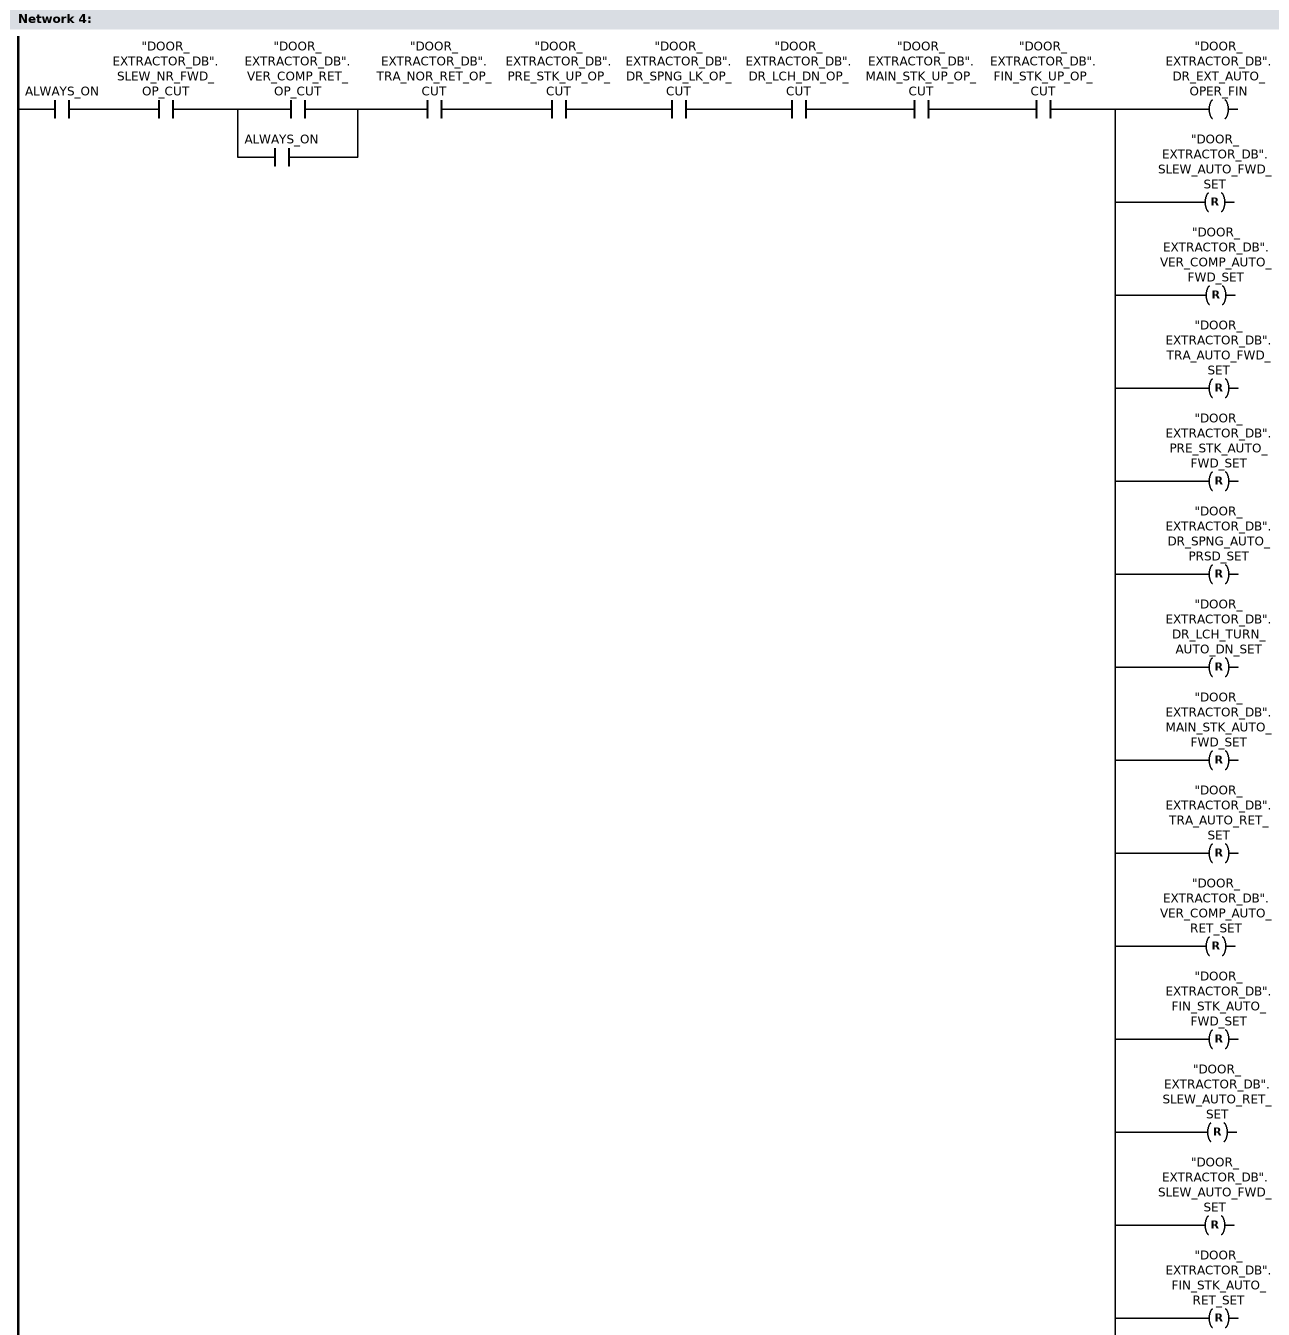
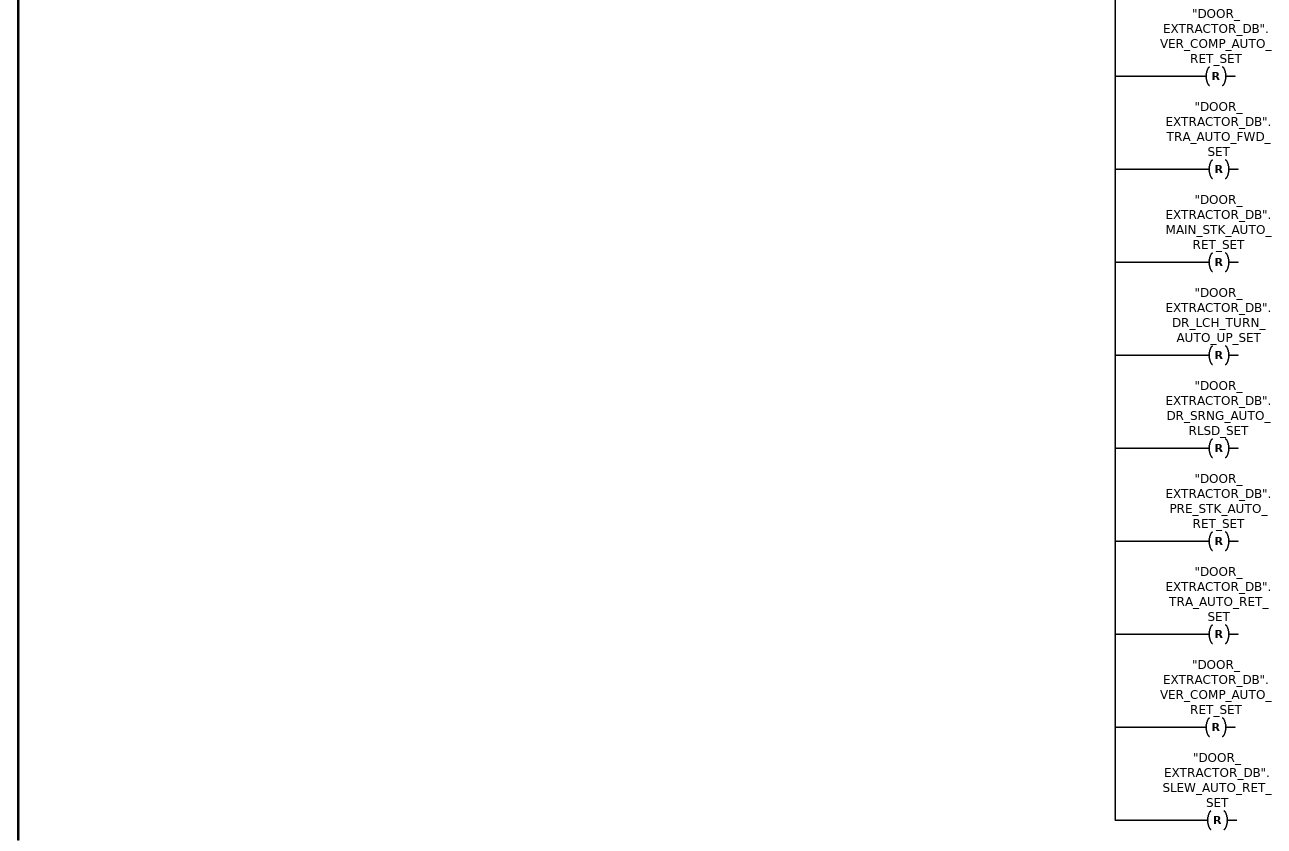
NETWORK
TITLE =
      A     "ALWAYS_ON";
      A     "DOOR_EXTRACTOR_DB".SLEW_NR_FWD_OP_CUT;
      A(;
      O     "DOOR_EXTRACTOR_DB".VER_COMP_RET_OP_CUT;
      O     "ALWAYS_ON";
      );
      A     "DOOR_EXTRACTOR_DB".TRA_NOR_RET_OP_CUT;
      A     "DOOR_EXTRACTOR_DB".PRE_STK_UP_OP_CUT;
      A     "DOOR_EXTRACTOR_DB".DR_SPNG_LK_OP_CUT;
      A     "DOOR_EXTRACTOR_DB".DR_LCH_DN_OP_CUT;
      A     "DOOR_EXTRACTOR_DB".MAIN_STK_UP_OP_CUT;
      A     "DOOR_EXTRACTOR_DB".FIN_STK_UP_OP_CUT;
      =     "DOOR_EXTRACTOR_DB".DR_EXT_AUTO_OPER_FIN;
      R     "DOOR_EXTRACTOR_DB".SLEW_AUTO_FWD_SET;
      R     "DOOR_EXTRACTOR_DB".VER_COMP_AUTO_FWD_SET;
      R     "DOOR_EXTRACTOR_DB".TRA_AUTO_FWD_SET;
      R     "DOOR_EXTRACTOR_DB".PRE_STK_AUTO_FWD_SET;
      R     "DOOR_EXTRACTOR_DB".DR_SPNG_AUTO_PRSD_SET;
      R     "DOOR_EXTRACTOR_DB".DR_LCH_TURN_AUTO_DN_SET;
      R     "DOOR_EXTRACTOR_DB".MAIN_STK_AUTO_FWD_SET;
      R     "DOOR_EXTRACTOR_DB".TRA_AUTO_RET_SET;
      R     "DOOR_EXTRACTOR_DB".VER_COMP_AUTO_RET_SET;
      R     "DOOR_EXTRACTOR_DB".FIN_STK_AUTO_FWD_SET;
      R     "DOOR_EXTRACTOR_DB".SLEW_AUTO_RET_SET;
      R     "DOOR_EXTRACTOR_DB".SLEW_AUTO_FWD_SET;
      R     "DOOR_EXTRACTOR_DB".FIN_STK_AUTO_RET_SET;
      R     "DOOR_EXTRACTOR_DB".VER_COMP_AUTO_RET_SET;
      R     "DOOR_EXTRACTOR_DB".TRA_AUTO_FWD_SET;
      R     "DOOR_EXTRACTOR_DB".MAIN_STK_AUTO_RET_SET;
      R     "DOOR_EXTRACTOR_DB".DR_LCH_TURN_AUTO_UP_SET;
      R     "DOOR_EXTRACTOR_DB".DR_SRNG_AUTO_RLSD_SET;
      R     "DOOR_EXTRACTOR_DB".PRE_STK_AUTO_RET_SET;
      R     "DOOR_EXTRACTOR_DB".TRA_AUTO_RET_SET;
      R     "DOOR_EXTRACTOR_DB".VER_COMP_AUTO_RET_SET;
      R     "DOOR_EXTRACTOR_DB".SLEW_AUTO_RET_SET;
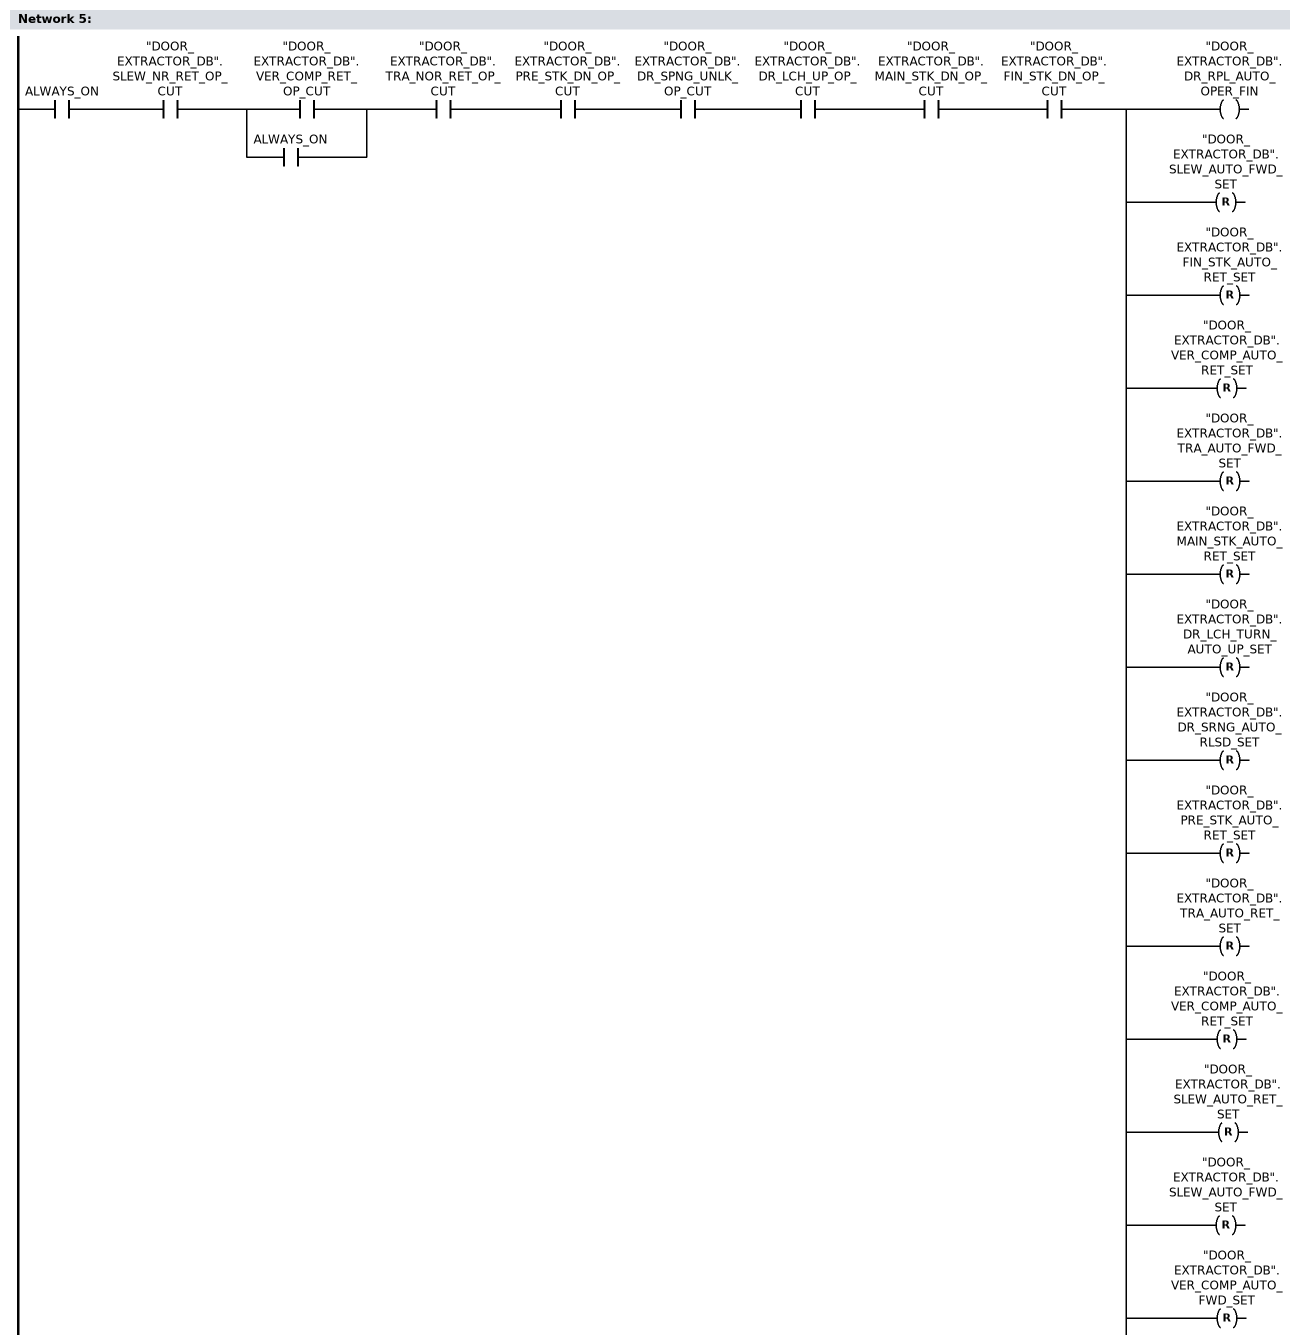
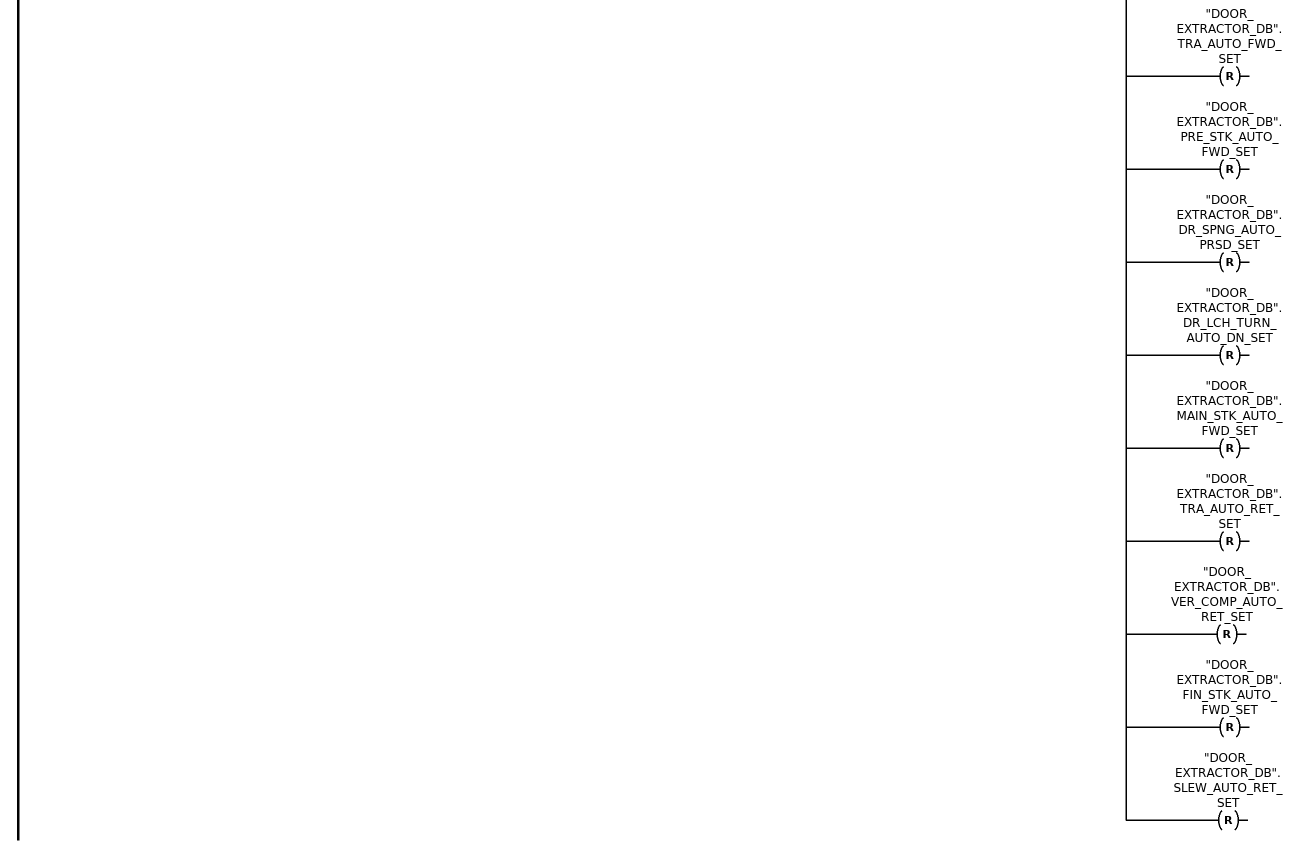
NETWORK
TITLE =
      A     "ALWAYS_ON";
      A     "DOOR_EXTRACTOR_DB".SLEW_NR_RET_OP_CUT;
      A(;
      O     "DOOR_EXTRACTOR_DB".VER_COMP_RET_OP_CUT;
      O     "ALWAYS_ON";
      );
      A     "DOOR_EXTRACTOR_DB".TRA_NOR_RET_OP_CUT;
      A     "DOOR_EXTRACTOR_DB".PRE_STK_DN_OP_CUT;
      A     "DOOR_EXTRACTOR_DB".DR_SPNG_UNLK_OP_CUT;
      A     "DOOR_EXTRACTOR_DB".DR_LCH_UP_OP_CUT;
      A     "DOOR_EXTRACTOR_DB".MAIN_STK_DN_OP_CUT;
      A     "DOOR_EXTRACTOR_DB".FIN_STK_DN_OP_CUT;
      =     "DOOR_EXTRACTOR_DB".DR_RPL_AUTO_OPER_FIN;
      R     "DOOR_EXTRACTOR_DB".SLEW_AUTO_FWD_SET;
      R     "DOOR_EXTRACTOR_DB".FIN_STK_AUTO_RET_SET;
      R     "DOOR_EXTRACTOR_DB".VER_COMP_AUTO_RET_SET;
      R     "DOOR_EXTRACTOR_DB".TRA_AUTO_FWD_SET;
      R     "DOOR_EXTRACTOR_DB".MAIN_STK_AUTO_RET_SET;
      R     "DOOR_EXTRACTOR_DB".DR_LCH_TURN_AUTO_UP_SET;
      R     "DOOR_EXTRACTOR_DB".DR_SRNG_AUTO_RLSD_SET;
      R     "DOOR_EXTRACTOR_DB".PRE_STK_AUTO_RET_SET;
      R     "DOOR_EXTRACTOR_DB".TRA_AUTO_RET_SET;
      R     "DOOR_EXTRACTOR_DB".VER_COMP_AUTO_RET_SET;
      R     "DOOR_EXTRACTOR_DB".SLEW_AUTO_RET_SET;
      R     "DOOR_EXTRACTOR_DB".SLEW_AUTO_FWD_SET;
      R     "DOOR_EXTRACTOR_DB".VER_COMP_AUTO_FWD_SET;
      R     "DOOR_EXTRACTOR_DB".TRA_AUTO_FWD_SET;
      R     "DOOR_EXTRACTOR_DB".PRE_STK_AUTO_FWD_SET;
      R     "DOOR_EXTRACTOR_DB".DR_SPNG_AUTO_PRSD_SET;
      R     "DOOR_EXTRACTOR_DB".DR_LCH_TURN_AUTO_DN_SET;
      R     "DOOR_EXTRACTOR_DB".MAIN_STK_AUTO_FWD_SET;
      R     "DOOR_EXTRACTOR_DB".TRA_AUTO_RET_SET;
      R     "DOOR_EXTRACTOR_DB".VER_COMP_AUTO_RET_SET;
      R     "DOOR_EXTRACTOR_DB".FIN_STK_AUTO_FWD_SET;
      R     "DOOR_EXTRACTOR_DB".SLEW_AUTO_RET_SET;
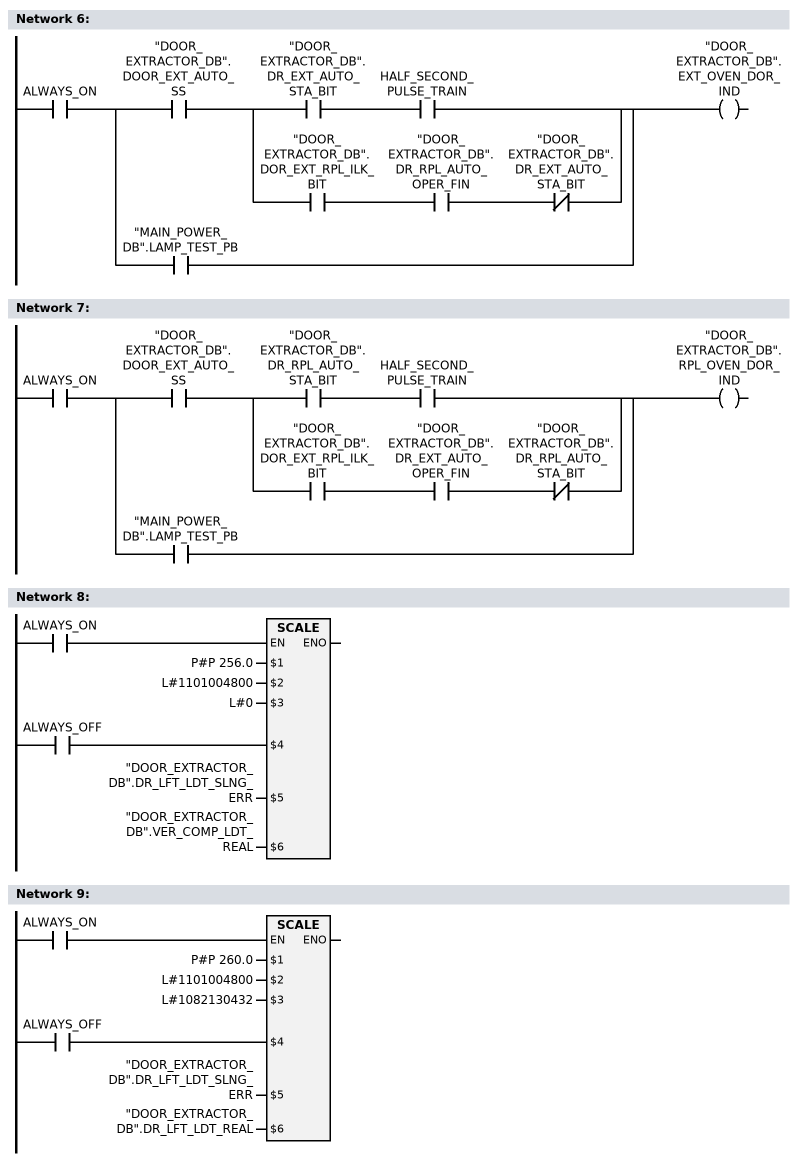
NETWORK
TITLE =
      A     "ALWAYS_ON";
      A(;
      A     "DOOR_EXTRACTOR_DB".DOOR_EXT_AUTO_SS;
      A(;
      A     "DOOR_EXTRACTOR_DB".DR_EXT_AUTO_STA_BIT;
      A     "HALF_SECOND_PULSE_TRAIN";
      O;
      A     "DOOR_EXTRACTOR_DB".DOR_EXT_RPL_ILK_BIT;
      A     "DOOR_EXTRACTOR_DB".DR_RPL_AUTO_OPER_FIN;
      AN    "DOOR_EXTRACTOR_DB".DR_EXT_AUTO_STA_BIT;
      );
      O     "MAIN_POWER_DB".LAMP_TEST_PB;
      );
      =     "DOOR_EXTRACTOR_DB".EXT_OVEN_DOR_IND;
NETWORK
TITLE =
      A     "ALWAYS_ON";
      A(;
      A     "DOOR_EXTRACTOR_DB".DOOR_EXT_AUTO_SS;
      A(;
      A     "DOOR_EXTRACTOR_DB".DR_RPL_AUTO_STA_BIT;
      A     "HALF_SECOND_PULSE_TRAIN";
      O;
      A     "DOOR_EXTRACTOR_DB".DOR_EXT_RPL_ILK_BIT;
      A     "DOOR_EXTRACTOR_DB".DR_EXT_AUTO_OPER_FIN;
      AN    "DOOR_EXTRACTOR_DB".DR_RPL_AUTO_STA_BIT;
      );
      O     "MAIN_POWER_DB".LAMP_TEST_PB;
      );
      =     "DOOR_EXTRACTOR_DB".RPL_OVEN_DOR_IND;
NETWORK
TITLE =
      A     "ALWAYS_OFF";
      =     L 0.0;
      BLD   103;
      A     "ALWAYS_ON";
      JNB   _001;
      CALL  "SCALE" (
           $1                       := P#P 256.0,
           $2                       := L#1101004800,
           $3                       := L#0,
           $4                       := L 0.0,
           $5                       := "DOOR_EXTRACTOR_DB".DR_LFT_LDT_SLNG_ERR,
           $6                       := "DOOR_EXTRACTOR_DB".VER_COMP_LDT_REAL);
_001: NOP   0;
NETWORK
TITLE =
      A     "ALWAYS_OFF";
      =     L 0.0;
      BLD   103;
      A     "ALWAYS_ON";
      JNB   _002;
      CALL  "SCALE" (
           $1                       := P#P 260.0,
           $2                       := L#1101004800,
           $3                       := L#1082130432,
           $4                       := L 0.0,
           $5                       := "DOOR_EXTRACTOR_DB".DR_LFT_LDT_SLNG_ERR,
           $6                       := "DOOR_EXTRACTOR_DB".DR_LFT_LDT_REAL);
_002: NOP   0;
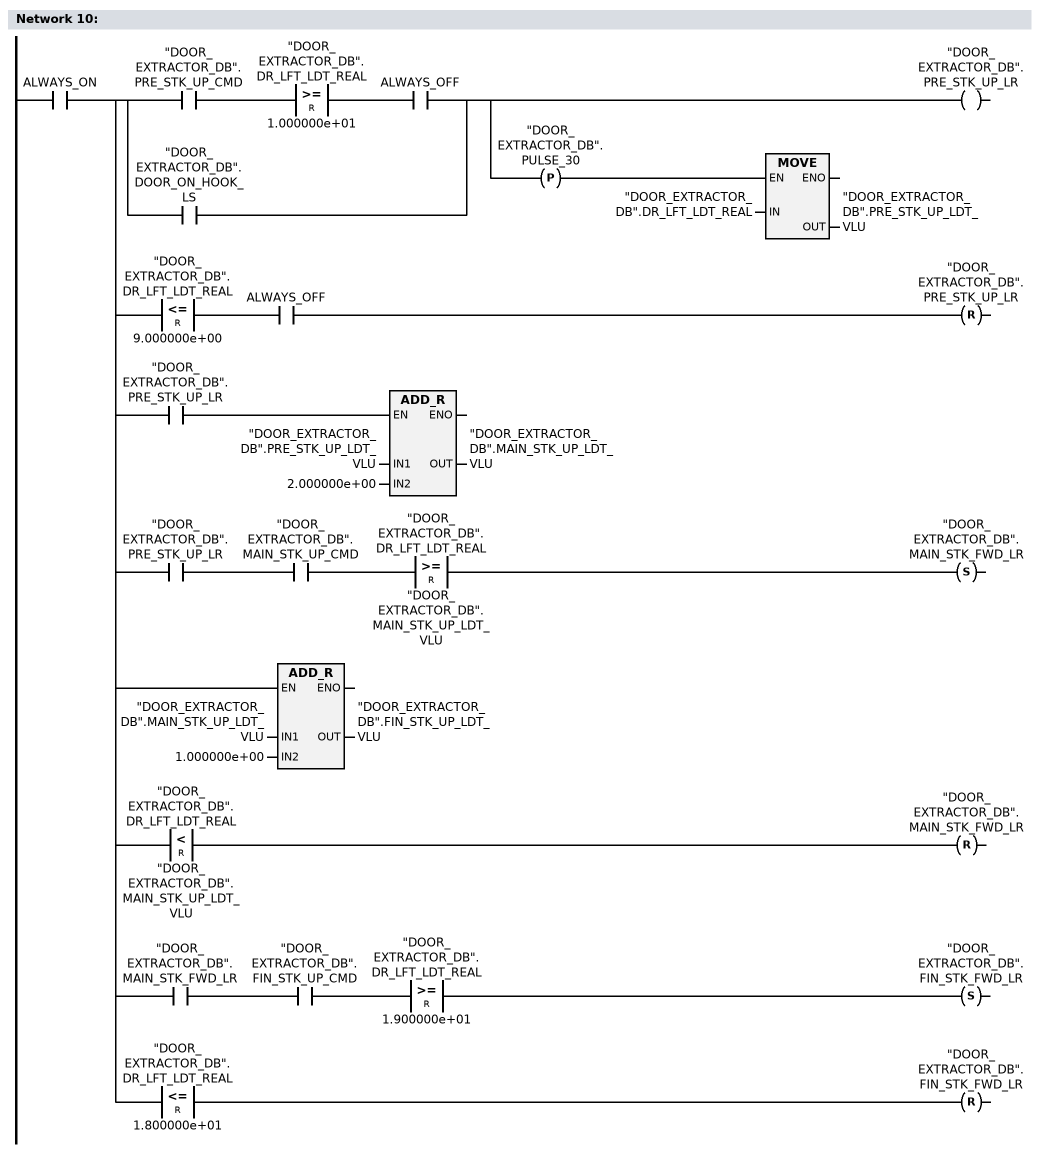
NETWORK
TITLE =
      A     "ALWAYS_ON";
      =     L 0.0;
      A     L 0.0;
      A(;
      A     "DOOR_EXTRACTOR_DB".PRE_STK_UP_CMD;
      A(;
      L     "DOOR_EXTRACTOR_DB".DR_LFT_LDT_REAL;
      L     1.000000e+01;
      >=R;
      );
      A     "ALWAYS_OFF";
      O     "DOOR_EXTRACTOR_DB".DOOR_ON_HOOK_LS;
      );
      =     L 0.1;
      A     L 0.1;
      BLD   102;
      =     "DOOR_EXTRACTOR_DB".PRE_STK_UP_LR;
      A     L 0.1;
      FP    "DOOR_EXTRACTOR_DB".PULSE_30;
      JNB   _003;
      L     "DOOR_EXTRACTOR_DB".DR_LFT_LDT_REAL;
      T     "DOOR_EXTRACTOR_DB".PRE_STK_UP_LDT_VLU;
_003: NOP   0;
      A     L 0.0;
      A(;
      L     "DOOR_EXTRACTOR_DB".DR_LFT_LDT_REAL;
      L     9.000000e+00;
      <=R;
      );
      A     "ALWAYS_OFF";
      R     "DOOR_EXTRACTOR_DB".PRE_STK_UP_LR;
      A     L 0.0;
      A     "DOOR_EXTRACTOR_DB".PRE_STK_UP_LR;
      JNB   _004;
      L     "DOOR_EXTRACTOR_DB".PRE_STK_UP_LDT_VLU;
      L     2.000000e+00;
      +R;
      T     "DOOR_EXTRACTOR_DB".MAIN_STK_UP_LDT_VLU;
_004: NOP   0;
      A     L 0.0;
      A     "DOOR_EXTRACTOR_DB".PRE_STK_UP_LR;
      A     "DOOR_EXTRACTOR_DB".MAIN_STK_UP_CMD;
      A(;
      L     "DOOR_EXTRACTOR_DB".DR_LFT_LDT_REAL;
      L     "DOOR_EXTRACTOR_DB".MAIN_STK_UP_LDT_VLU;
      >=R;
      );
      S     "DOOR_EXTRACTOR_DB".MAIN_STK_FWD_LR;
      A     L 0.0;
      JNB   _005;
      L     "DOOR_EXTRACTOR_DB".MAIN_STK_UP_LDT_VLU;
      L     1.000000e+00;
      +R;
      T     "DOOR_EXTRACTOR_DB".FIN_STK_UP_LDT_VLU;
_005: NOP   0;
      A     L 0.0;
      A(;
      L     "DOOR_EXTRACTOR_DB".DR_LFT_LDT_REAL;
      L     "DOOR_EXTRACTOR_DB".MAIN_STK_UP_LDT_VLU;
      <R;
      );
      R     "DOOR_EXTRACTOR_DB".MAIN_STK_FWD_LR;
      A     L 0.0;
      A     "DOOR_EXTRACTOR_DB".MAIN_STK_FWD_LR;
      A     "DOOR_EXTRACTOR_DB".FIN_STK_UP_CMD;
      A(;
      L     "DOOR_EXTRACTOR_DB".DR_LFT_LDT_REAL;
      L     1.900000e+01;
      >=R;
      );
      S     "DOOR_EXTRACTOR_DB".FIN_STK_FWD_LR;
      A     L 0.0;
      A(;
      L     "DOOR_EXTRACTOR_DB".DR_LFT_LDT_REAL;
      L     1.800000e+01;
      <=R;
      );
      R     "DOOR_EXTRACTOR_DB".FIN_STK_FWD_LR;
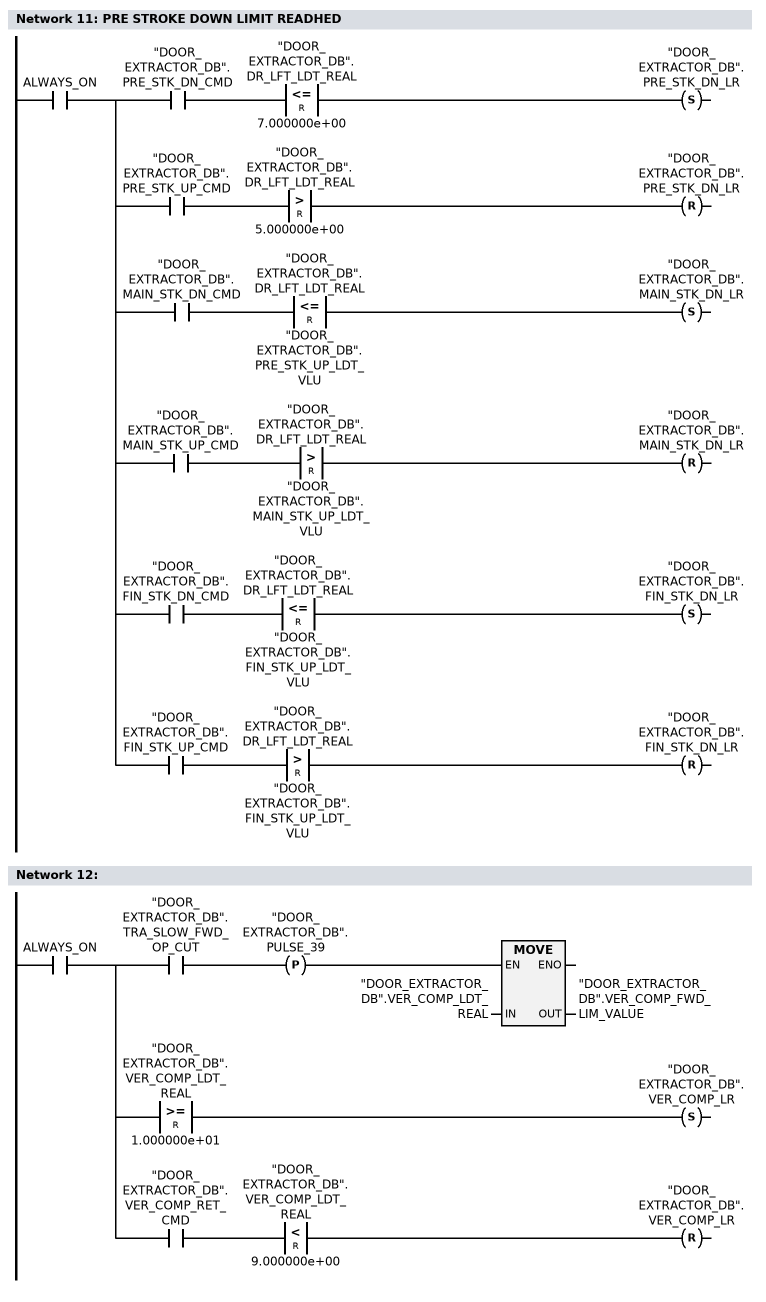
NETWORK
TITLE = PRE STROKE DOWN LIMIT READHED
      A     "ALWAYS_ON";
      =     L 0.0;
      A     L 0.0;
      A     "DOOR_EXTRACTOR_DB".PRE_STK_DN_CMD;
      A(;
      L     "DOOR_EXTRACTOR_DB".DR_LFT_LDT_REAL;
      L     7.000000e+00;
      <=R;
      );
      S     "DOOR_EXTRACTOR_DB".PRE_STK_DN_LR;
      A     L 0.0;
      A     "DOOR_EXTRACTOR_DB".PRE_STK_UP_CMD;
      A(;
      L     "DOOR_EXTRACTOR_DB".DR_LFT_LDT_REAL;
      L     5.000000e+00;
      >R;
      );
      R     "DOOR_EXTRACTOR_DB".PRE_STK_DN_LR;
      A     L 0.0;
      A     "DOOR_EXTRACTOR_DB".MAIN_STK_DN_CMD;
      A(;
      L     "DOOR_EXTRACTOR_DB".DR_LFT_LDT_REAL;
      L     "DOOR_EXTRACTOR_DB".PRE_STK_UP_LDT_VLU;
      <=R;
      );
      S     "DOOR_EXTRACTOR_DB".MAIN_STK_DN_LR;
      A     L 0.0;
      A     "DOOR_EXTRACTOR_DB".MAIN_STK_UP_CMD;
      A(;
      L     "DOOR_EXTRACTOR_DB".DR_LFT_LDT_REAL;
      L     "DOOR_EXTRACTOR_DB".MAIN_STK_UP_LDT_VLU;
      >R;
      );
      R     "DOOR_EXTRACTOR_DB".MAIN_STK_DN_LR;
      A     L 0.0;
      A     "DOOR_EXTRACTOR_DB".FIN_STK_DN_CMD;
      A(;
      L     "DOOR_EXTRACTOR_DB".DR_LFT_LDT_REAL;
      L     "DOOR_EXTRACTOR_DB".FIN_STK_UP_LDT_VLU;
      <=R;
      );
      S     "DOOR_EXTRACTOR_DB".FIN_STK_DN_LR;
      A     L 0.0;
      A     "DOOR_EXTRACTOR_DB".FIN_STK_UP_CMD;
      A(;
      L     "DOOR_EXTRACTOR_DB".DR_LFT_LDT_REAL;
      L     "DOOR_EXTRACTOR_DB".FIN_STK_UP_LDT_VLU;
      >R;
      );
      R     "DOOR_EXTRACTOR_DB".FIN_STK_DN_LR;
NETWORK
TITLE =
      A     "ALWAYS_ON";
      =     L 0.0;
      A     L 0.0;
      A     "DOOR_EXTRACTOR_DB".TRA_SLOW_FWD_OP_CUT;
      FP    "DOOR_EXTRACTOR_DB".PULSE_39;
      JNB   _006;
      L     "DOOR_EXTRACTOR_DB".VER_COMP_LDT_REAL;
      T     "DOOR_EXTRACTOR_DB".VER_COMP_FWD_LIM_VALUE;
_006: NOP   0;
      A     L 0.0;
      A(;
      L     "DOOR_EXTRACTOR_DB".VER_COMP_LDT_REAL;
      L     1.000000e+01;
      >=R;
      );
      S     "DOOR_EXTRACTOR_DB".VER_COMP_LR;
      A     L 0.0;
      A     "DOOR_EXTRACTOR_DB".VER_COMP_RET_CMD;
      A(;
      L     "DOOR_EXTRACTOR_DB".VER_COMP_LDT_REAL;
      L     9.000000e+00;
      <R;
      );
      R     "DOOR_EXTRACTOR_DB".VER_COMP_LR;
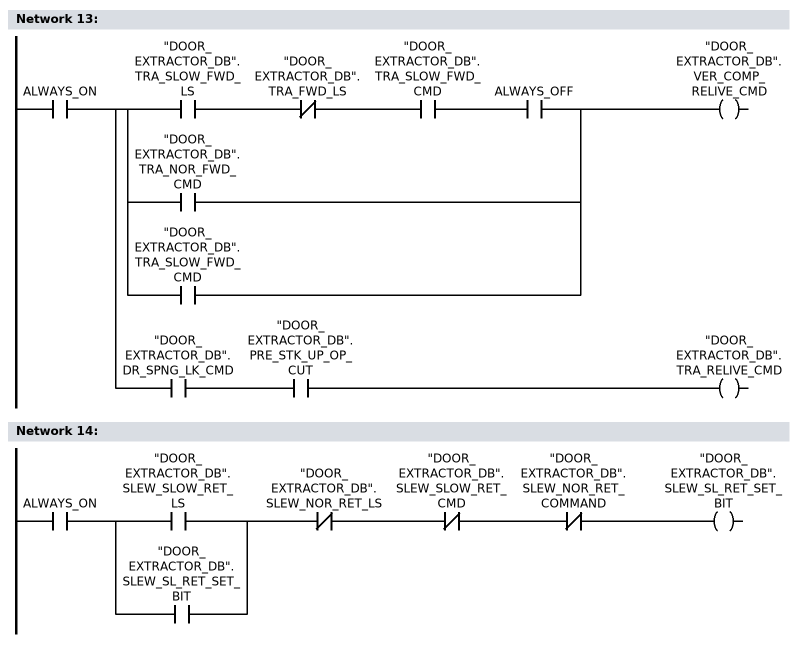
NETWORK
TITLE =
      A     "ALWAYS_ON";
      =     L 0.0;
      A     L 0.0;
      A(;
      A     "DOOR_EXTRACTOR_DB".TRA_SLOW_FWD_LS;
      AN    "DOOR_EXTRACTOR_DB".TRA_FWD_LS;
      A     "DOOR_EXTRACTOR_DB".TRA_SLOW_FWD_CMD;
      A     "ALWAYS_OFF";
      O     "DOOR_EXTRACTOR_DB".TRA_NOR_FWD_CMD;
      O     "DOOR_EXTRACTOR_DB".TRA_SLOW_FWD_CMD;
      );
      =     "DOOR_EXTRACTOR_DB".VER_COMP_RELIVE_CMD;
      A     L 0.0;
      A     "DOOR_EXTRACTOR_DB".DR_SPNG_LK_CMD;
      A     "DOOR_EXTRACTOR_DB".PRE_STK_UP_OP_CUT;
      =     "DOOR_EXTRACTOR_DB".TRA_RELIVE_CMD;
NETWORK
TITLE =
      A     "ALWAYS_ON";
      A(;
      O     "DOOR_EXTRACTOR_DB".SLEW_SLOW_RET_LS;
      O     "DOOR_EXTRACTOR_DB".SLEW_SL_RET_SET_BIT;
      );
      AN    "DOOR_EXTRACTOR_DB".SLEW_NOR_RET_LS;
      AN    "DOOR_EXTRACTOR_DB".SLEW_SLOW_RET_CMD;
      AN    "DOOR_EXTRACTOR_DB".SLEW_NOR_RET_COMMAND;
      =     "DOOR_EXTRACTOR_DB".SLEW_SL_RET_SET_BIT;
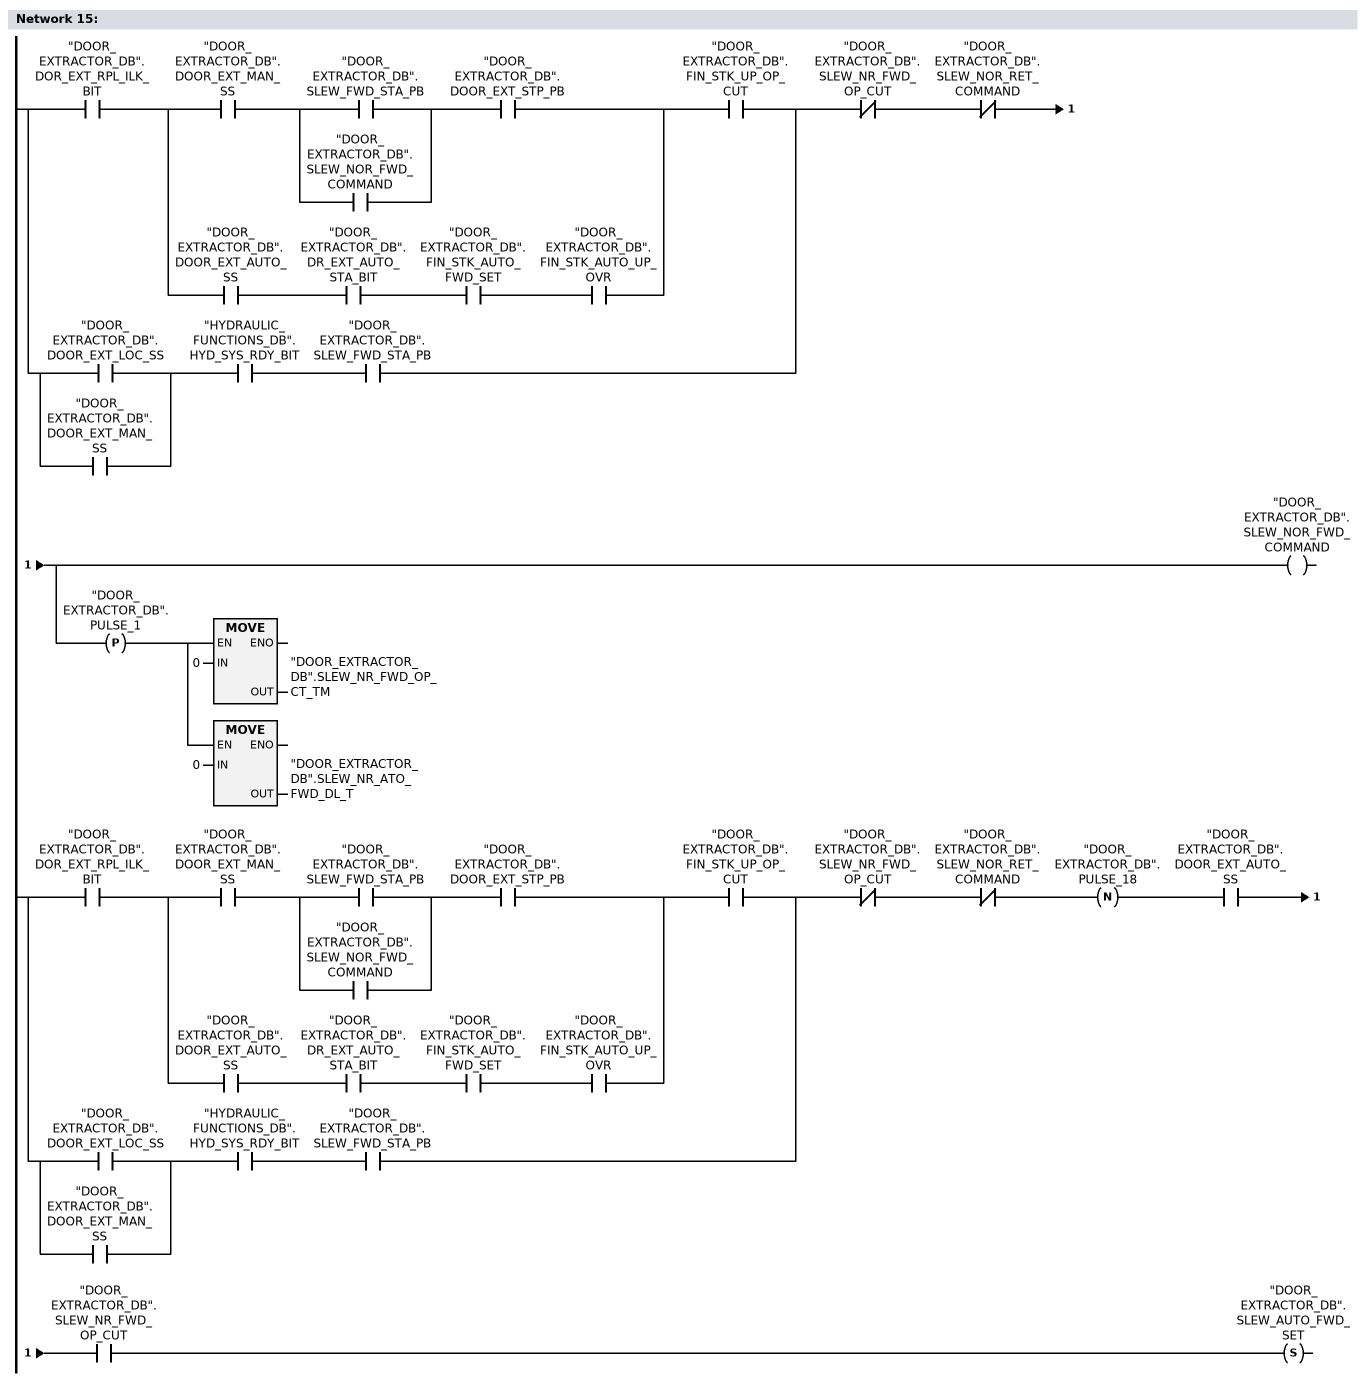
NETWORK
TITLE =
      A(;
      A     "DOOR_EXTRACTOR_DB".DOR_EXT_RPL_ILK_BIT;
      A(;
      A     "DOOR_EXTRACTOR_DB".DOOR_EXT_MAN_SS;
      A(;
      O     "DOOR_EXTRACTOR_DB".SLEW_FWD_STA_PB;
      O     "DOOR_EXTRACTOR_DB".SLEW_NOR_FWD_COMMAND;
      );
      A     "DOOR_EXTRACTOR_DB".DOOR_EXT_STP_PB;
      O;
      A     "DOOR_EXTRACTOR_DB".DOOR_EXT_AUTO_SS;
      A     "DOOR_EXTRACTOR_DB".DR_EXT_AUTO_STA_BIT;
      A     "DOOR_EXTRACTOR_DB".FIN_STK_AUTO_FWD_SET;
      A     "DOOR_EXTRACTOR_DB".FIN_STK_AUTO_UP_OVR;
      );
      A     "DOOR_EXTRACTOR_DB".FIN_STK_UP_OP_CUT;
      O;
      A(;
      O     "DOOR_EXTRACTOR_DB".DOOR_EXT_LOC_SS;
      O     "DOOR_EXTRACTOR_DB".DOOR_EXT_MAN_SS;
      );
      A     "HYDRAULIC_FUNCTIONS_DB".HYD_SYS_RDY_BIT;
      A     "DOOR_EXTRACTOR_DB".SLEW_FWD_STA_PB;
      );
      AN    "DOOR_EXTRACTOR_DB".SLEW_NR_FWD_OP_CUT;
      AN    "DOOR_EXTRACTOR_DB".SLEW_NOR_RET_COMMAND;
      =     L 0.0;
      A     L 0.0;
      BLD   102;
      =     "DOOR_EXTRACTOR_DB".SLEW_NOR_FWD_COMMAND;
      A(;
      A     L 0.0;
      FN    "DOOR_EXTRACTOR_DB".PULSE_18;
      );
      A     "DOOR_EXTRACTOR_DB".DOOR_EXT_AUTO_SS;
      A     "DOOR_EXTRACTOR_DB".SLEW_NR_FWD_OP_CUT;
      S     "DOOR_EXTRACTOR_DB".SLEW_AUTO_FWD_SET;
      A     L 0.0;
      FP    "DOOR_EXTRACTOR_DB".PULSE_1;
      =     L 0.1;
      A     L 0.1;
      JNB   _007;
      L     0;
      T     "DOOR_EXTRACTOR_DB".SLEW_NR_FWD_OP_CT_TM;
_007: NOP   0;
      A     L 0.1;
      JNB   _008;
      L     0;
      T     "DOOR_EXTRACTOR_DB".SLEW_NR_ATO_FWD_DL_T;
_008: NOP   0;
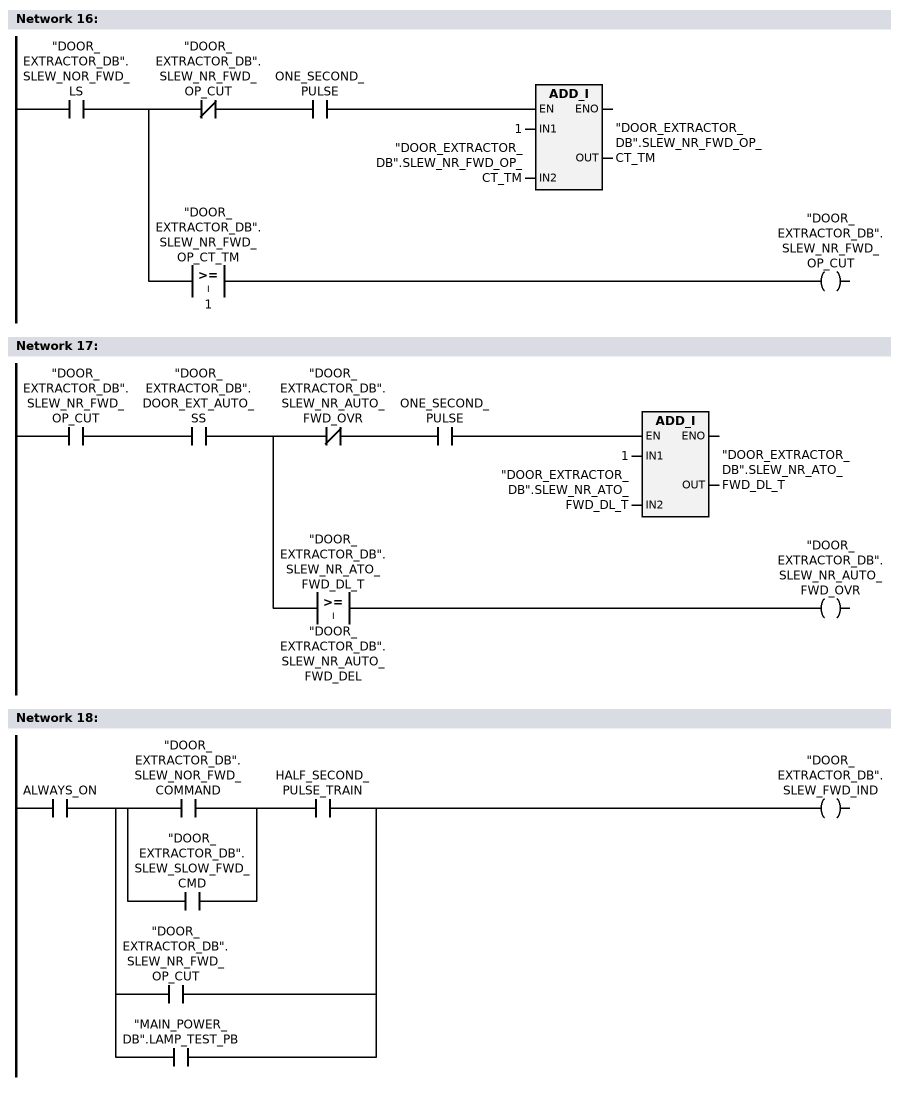
NETWORK
TITLE =
      A     "DOOR_EXTRACTOR_DB".SLEW_NOR_FWD_LS;
      =     L 0.0;
      A     L 0.0;
      AN    "DOOR_EXTRACTOR_DB".SLEW_NR_FWD_OP_CUT;
      A     "ONE_SECOND_PULSE";
      JNB   _009;
      L     1;
      L     "DOOR_EXTRACTOR_DB".SLEW_NR_FWD_OP_CT_TM;
      +I;
      T     "DOOR_EXTRACTOR_DB".SLEW_NR_FWD_OP_CT_TM;
_009: NOP   0;
      A     L 0.0;
      A(;
      L     "DOOR_EXTRACTOR_DB".SLEW_NR_FWD_OP_CT_TM;
      L     1;
      >=I;
      );
      =     "DOOR_EXTRACTOR_DB".SLEW_NR_FWD_OP_CUT;
NETWORK
TITLE =
      A     "DOOR_EXTRACTOR_DB".SLEW_NR_FWD_OP_CUT;
      A     "DOOR_EXTRACTOR_DB".DOOR_EXT_AUTO_SS;
      =     L 0.0;
      A     L 0.0;
      AN    "DOOR_EXTRACTOR_DB".SLEW_NR_AUTO_FWD_OVR;
      A     "ONE_SECOND_PULSE";
      JNB   _00a;
      L     1;
      L     "DOOR_EXTRACTOR_DB".SLEW_NR_ATO_FWD_DL_T;
      +I;
      T     "DOOR_EXTRACTOR_DB".SLEW_NR_ATO_FWD_DL_T;
_00a: NOP   0;
      A     L 0.0;
      A(;
      L     "DOOR_EXTRACTOR_DB".SLEW_NR_ATO_FWD_DL_T;
      L     "DOOR_EXTRACTOR_DB".SLEW_NR_AUTO_FWD_DEL;
      >=I;
      );
      =     "DOOR_EXTRACTOR_DB".SLEW_NR_AUTO_FWD_OVR;
NETWORK
TITLE =
      A     "ALWAYS_ON";
      A(;
      A(;
      O     "DOOR_EXTRACTOR_DB".SLEW_NOR_FWD_COMMAND;
      O     "DOOR_EXTRACTOR_DB".SLEW_SLOW_FWD_CMD;
      );
      A     "HALF_SECOND_PULSE_TRAIN";
      O     "DOOR_EXTRACTOR_DB".SLEW_NR_FWD_OP_CUT;
      O     "MAIN_POWER_DB".LAMP_TEST_PB;
      );
      =     "DOOR_EXTRACTOR_DB".SLEW_FWD_IND;
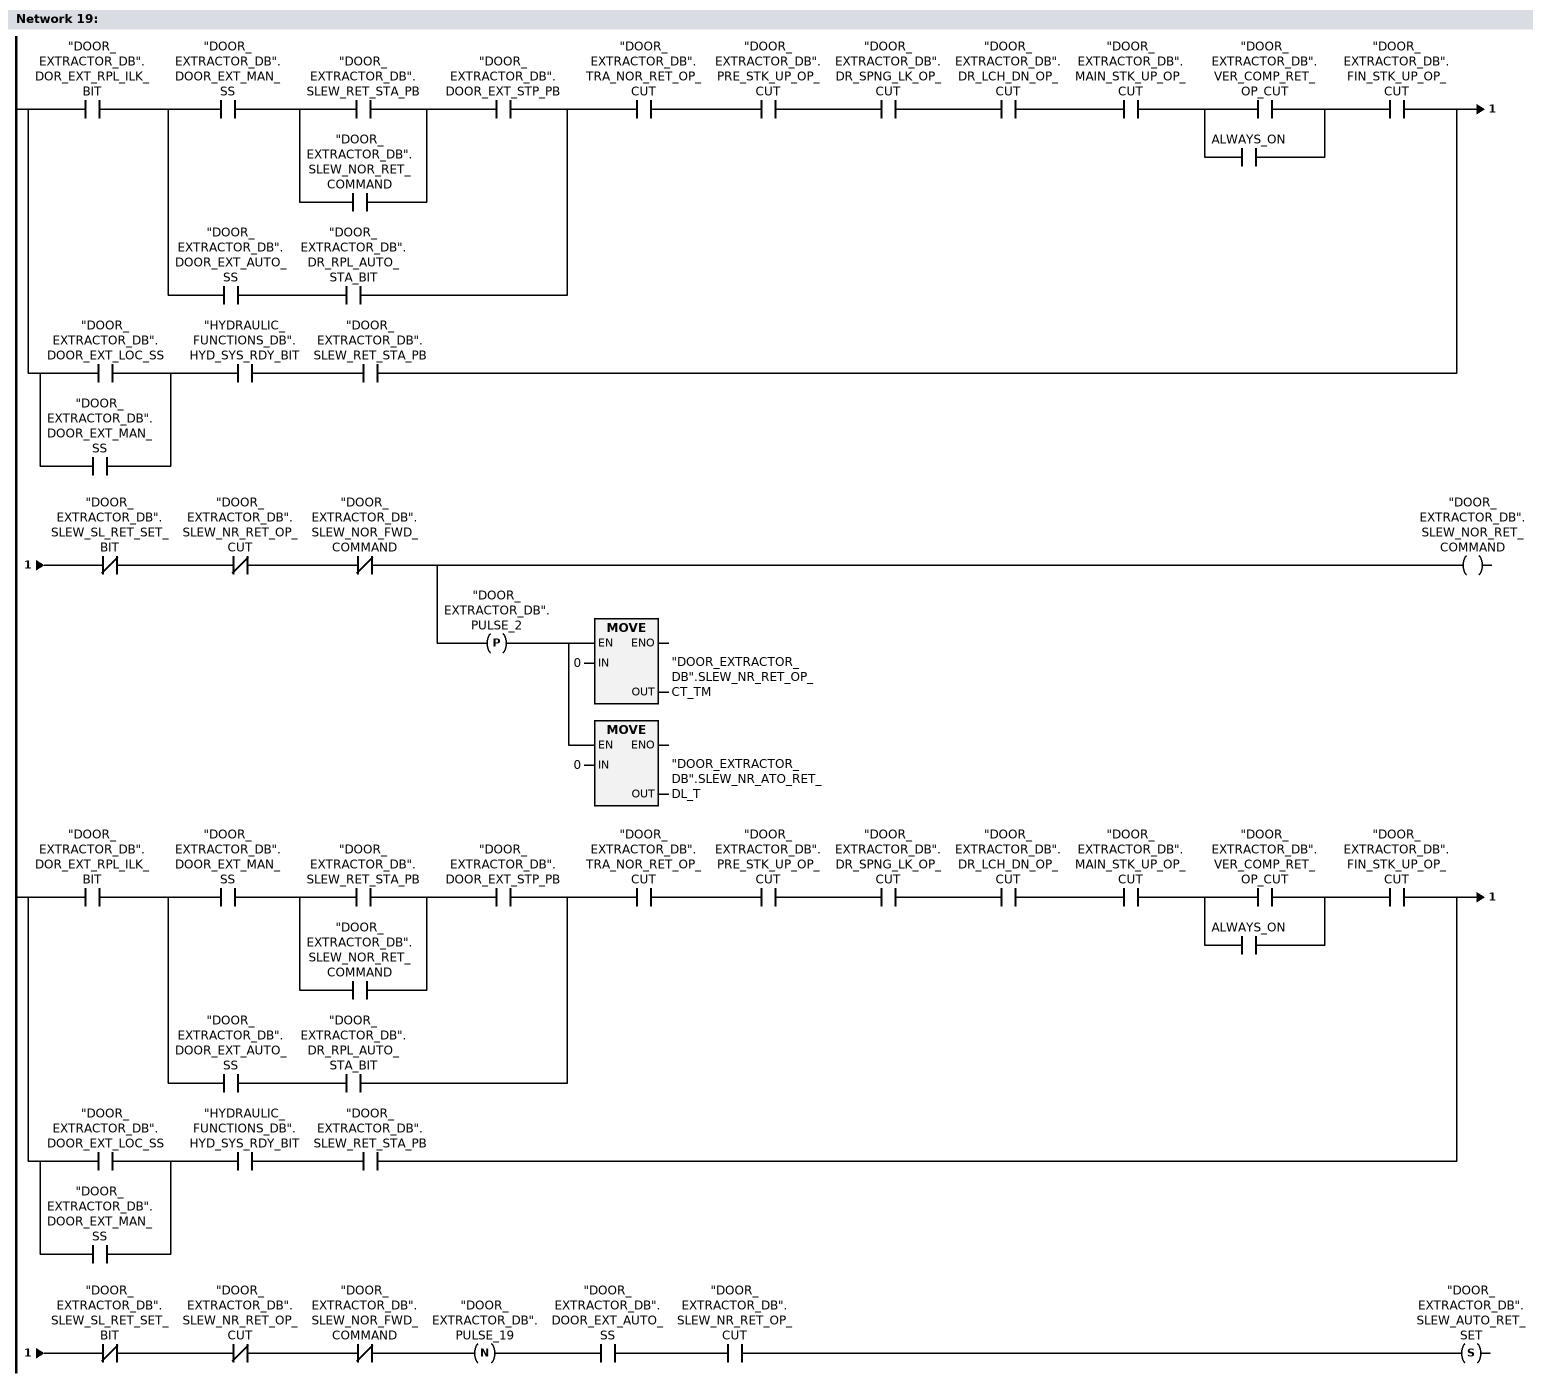
NETWORK
TITLE =
      A(;
      A     "DOOR_EXTRACTOR_DB".DOR_EXT_RPL_ILK_BIT;
      A(;
      A     "DOOR_EXTRACTOR_DB".DOOR_EXT_MAN_SS;
      A(;
      O     "DOOR_EXTRACTOR_DB".SLEW_RET_STA_PB;
      O     "DOOR_EXTRACTOR_DB".SLEW_NOR_RET_COMMAND;
      );
      A     "DOOR_EXTRACTOR_DB".DOOR_EXT_STP_PB;
      O;
      A     "DOOR_EXTRACTOR_DB".DOOR_EXT_AUTO_SS;
      A     "DOOR_EXTRACTOR_DB".DR_RPL_AUTO_STA_BIT;
      );
      A     "DOOR_EXTRACTOR_DB".TRA_NOR_RET_OP_CUT;
      A     "DOOR_EXTRACTOR_DB".PRE_STK_UP_OP_CUT;
      A     "DOOR_EXTRACTOR_DB".DR_SPNG_LK_OP_CUT;
      A     "DOOR_EXTRACTOR_DB".DR_LCH_DN_OP_CUT;
      A     "DOOR_EXTRACTOR_DB".MAIN_STK_UP_OP_CUT;
      A(;
      O     "DOOR_EXTRACTOR_DB".VER_COMP_RET_OP_CUT;
      O     "ALWAYS_ON";
      );
      A     "DOOR_EXTRACTOR_DB".FIN_STK_UP_OP_CUT;
      O;
      A(;
      O     "DOOR_EXTRACTOR_DB".DOOR_EXT_LOC_SS;
      O     "DOOR_EXTRACTOR_DB".DOOR_EXT_MAN_SS;
      );
      A     "HYDRAULIC_FUNCTIONS_DB".HYD_SYS_RDY_BIT;
      A     "DOOR_EXTRACTOR_DB".SLEW_RET_STA_PB;
      );
      AN    "DOOR_EXTRACTOR_DB".SLEW_SL_RET_SET_BIT;
      AN    "DOOR_EXTRACTOR_DB".SLEW_NR_RET_OP_CUT;
      AN    "DOOR_EXTRACTOR_DB".SLEW_NOR_FWD_COMMAND;
      =     L 0.0;
      A     L 0.0;
      BLD   102;
      =     "DOOR_EXTRACTOR_DB".SLEW_NOR_RET_COMMAND;
      A(;
      A     L 0.0;
      FN    "DOOR_EXTRACTOR_DB".PULSE_19;
      );
      A     "DOOR_EXTRACTOR_DB".DOOR_EXT_AUTO_SS;
      A     "DOOR_EXTRACTOR_DB".SLEW_NR_RET_OP_CUT;
      S     "DOOR_EXTRACTOR_DB".SLEW_AUTO_RET_SET;
      A     L 0.0;
      FP    "DOOR_EXTRACTOR_DB".PULSE_2;
      =     L 0.1;
      A     L 0.1;
      JNB   _00b;
      L     0;
      T     "DOOR_EXTRACTOR_DB".SLEW_NR_RET_OP_CT_TM;
_00b: NOP   0;
      A     L 0.1;
      JNB   _00c;
      L     0;
      T     "DOOR_EXTRACTOR_DB".SLEW_NR_ATO_RET_DL_T;
_00c: NOP   0;
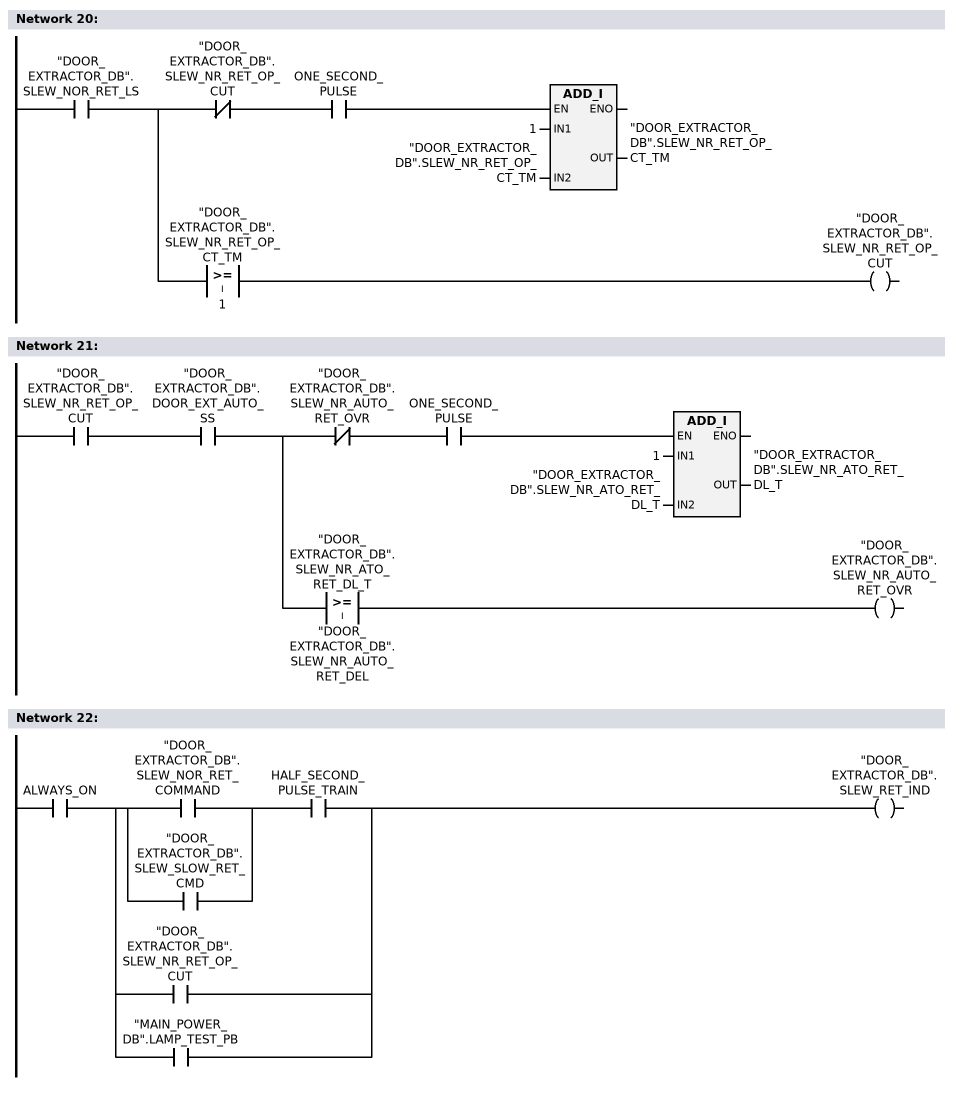
NETWORK
TITLE =
      A     "DOOR_EXTRACTOR_DB".SLEW_NOR_RET_LS;
      =     L 0.0;
      A     L 0.0;
      AN    "DOOR_EXTRACTOR_DB".SLEW_NR_RET_OP_CUT;
      A     "ONE_SECOND_PULSE";
      JNB   _00d;
      L     1;
      L     "DOOR_EXTRACTOR_DB".SLEW_NR_RET_OP_CT_TM;
      +I;
      T     "DOOR_EXTRACTOR_DB".SLEW_NR_RET_OP_CT_TM;
_00d: NOP   0;
      A     L 0.0;
      A(;
      L     "DOOR_EXTRACTOR_DB".SLEW_NR_RET_OP_CT_TM;
      L     1;
      >=I;
      );
      =     "DOOR_EXTRACTOR_DB".SLEW_NR_RET_OP_CUT;
NETWORK
TITLE =
      A     "DOOR_EXTRACTOR_DB".SLEW_NR_RET_OP_CUT;
      A     "DOOR_EXTRACTOR_DB".DOOR_EXT_AUTO_SS;
      =     L 0.0;
      A     L 0.0;
      AN    "DOOR_EXTRACTOR_DB".SLEW_NR_AUTO_RET_OVR;
      A     "ONE_SECOND_PULSE";
      JNB   _00e;
      L     1;
      L     "DOOR_EXTRACTOR_DB".SLEW_NR_ATO_RET_DL_T;
      +I;
      T     "DOOR_EXTRACTOR_DB".SLEW_NR_ATO_RET_DL_T;
_00e: NOP   0;
      A     L 0.0;
      A(;
      L     "DOOR_EXTRACTOR_DB".SLEW_NR_ATO_RET_DL_T;
      L     "DOOR_EXTRACTOR_DB".SLEW_NR_AUTO_RET_DEL;
      >=I;
      );
      =     "DOOR_EXTRACTOR_DB".SLEW_NR_AUTO_RET_OVR;
NETWORK
TITLE =
      A     "ALWAYS_ON";
      A(;
      A(;
      O     "DOOR_EXTRACTOR_DB".SLEW_NOR_RET_COMMAND;
      O     "DOOR_EXTRACTOR_DB".SLEW_SLOW_RET_CMD;
      );
      A     "HALF_SECOND_PULSE_TRAIN";
      O     "DOOR_EXTRACTOR_DB".SLEW_NR_RET_OP_CUT;
      O     "MAIN_POWER_DB".LAMP_TEST_PB;
      );
      =     "DOOR_EXTRACTOR_DB".SLEW_RET_IND;
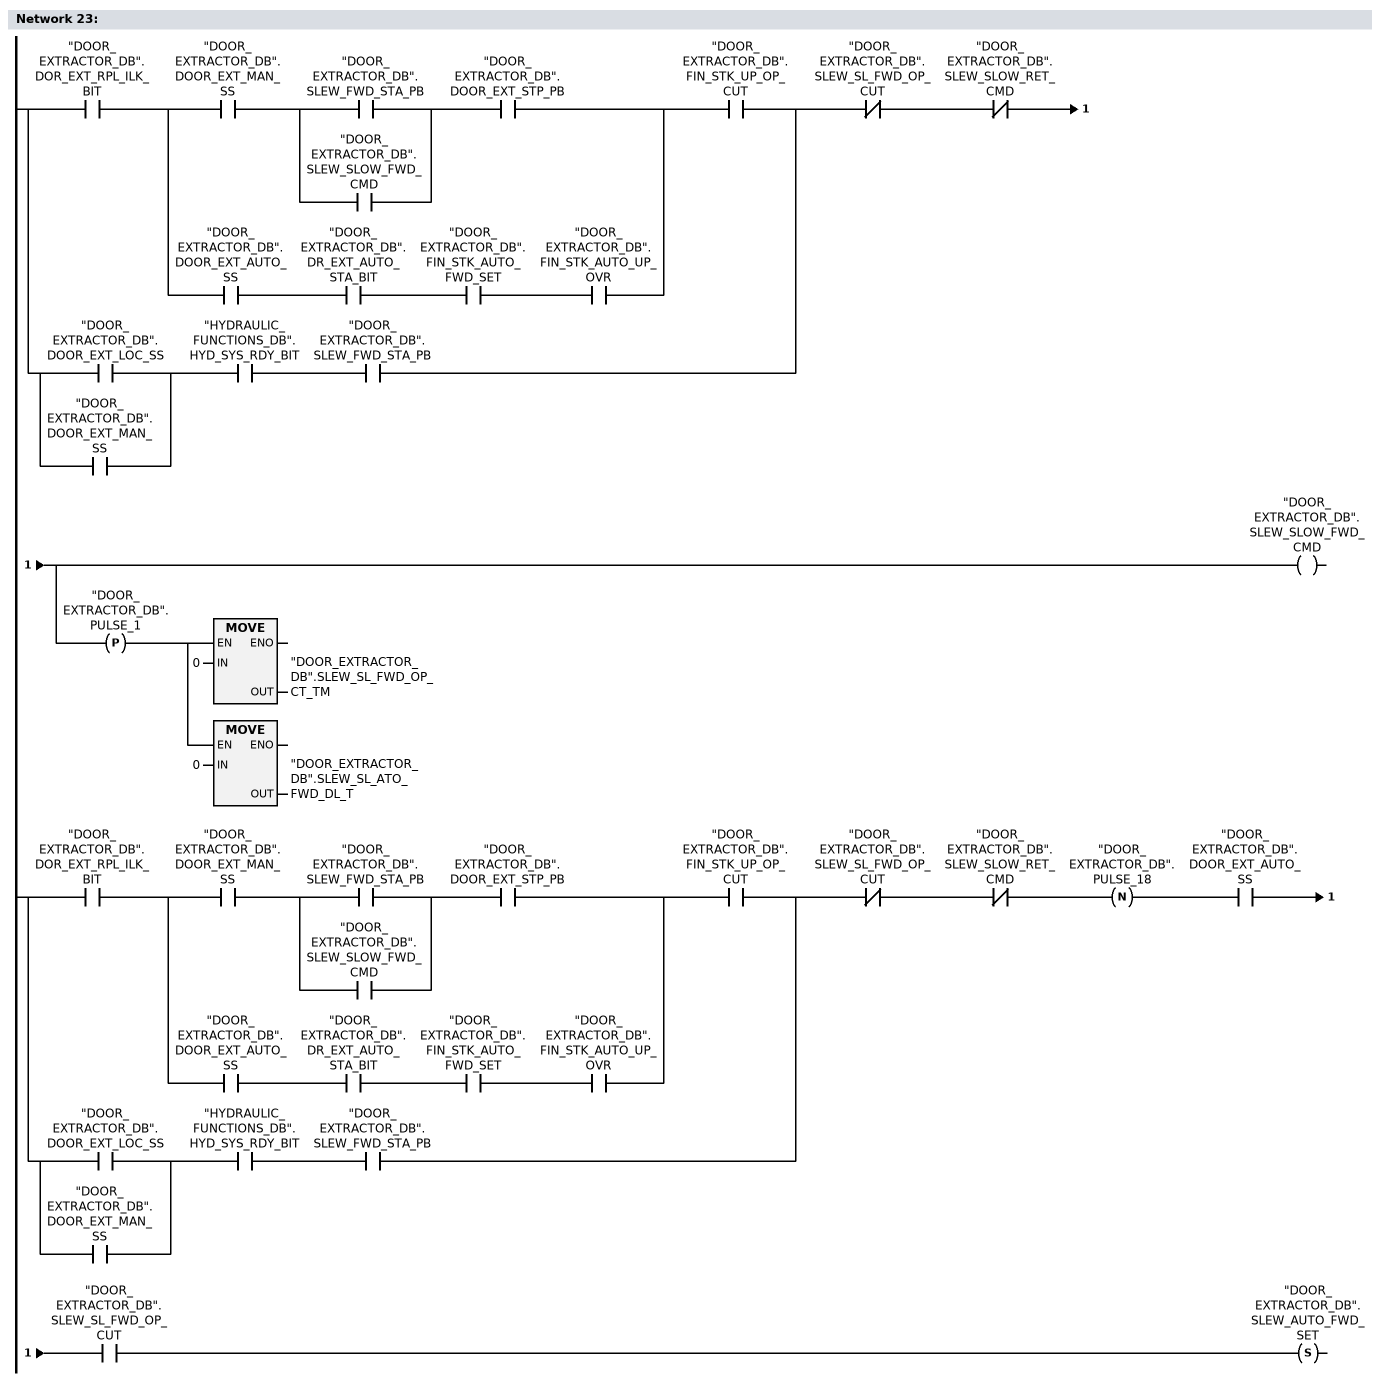
NETWORK
TITLE =
      A(;
      A     "DOOR_EXTRACTOR_DB".DOR_EXT_RPL_ILK_BIT;
      A(;
      A     "DOOR_EXTRACTOR_DB".DOOR_EXT_MAN_SS;
      A(;
      O     "DOOR_EXTRACTOR_DB".SLEW_FWD_STA_PB;
      O     "DOOR_EXTRACTOR_DB".SLEW_SLOW_FWD_CMD;
      );
      A     "DOOR_EXTRACTOR_DB".DOOR_EXT_STP_PB;
      O;
      A     "DOOR_EXTRACTOR_DB".DOOR_EXT_AUTO_SS;
      A     "DOOR_EXTRACTOR_DB".DR_EXT_AUTO_STA_BIT;
      A     "DOOR_EXTRACTOR_DB".FIN_STK_AUTO_FWD_SET;
      A     "DOOR_EXTRACTOR_DB".FIN_STK_AUTO_UP_OVR;
      );
      A     "DOOR_EXTRACTOR_DB".FIN_STK_UP_OP_CUT;
      O;
      A(;
      O     "DOOR_EXTRACTOR_DB".DOOR_EXT_LOC_SS;
      O     "DOOR_EXTRACTOR_DB".DOOR_EXT_MAN_SS;
      );
      A     "HYDRAULIC_FUNCTIONS_DB".HYD_SYS_RDY_BIT;
      A     "DOOR_EXTRACTOR_DB".SLEW_FWD_STA_PB;
      );
      AN    "DOOR_EXTRACTOR_DB".SLEW_SL_FWD_OP_CUT;
      AN    "DOOR_EXTRACTOR_DB".SLEW_SLOW_RET_CMD;
      =     L 0.0;
      A     L 0.0;
      BLD   102;
      =     "DOOR_EXTRACTOR_DB".SLEW_SLOW_FWD_CMD;
      A(;
      A     L 0.0;
      FN    "DOOR_EXTRACTOR_DB".PULSE_18;
      );
      A     "DOOR_EXTRACTOR_DB".DOOR_EXT_AUTO_SS;
      A     "DOOR_EXTRACTOR_DB".SLEW_SL_FWD_OP_CUT;
      S     "DOOR_EXTRACTOR_DB".SLEW_AUTO_FWD_SET;
      A     L 0.0;
      FP    "DOOR_EXTRACTOR_DB".PULSE_1;
      =     L 0.1;
      A     L 0.1;
      JNB   _00f;
      L     0;
      T     "DOOR_EXTRACTOR_DB".SLEW_SL_FWD_OP_CT_TM;
_00f: NOP   0;
      A     L 0.1;
      JNB   _010;
      L     0;
      T     "DOOR_EXTRACTOR_DB".SLEW_SL_ATO_FWD_DL_T;
_010: NOP   0;
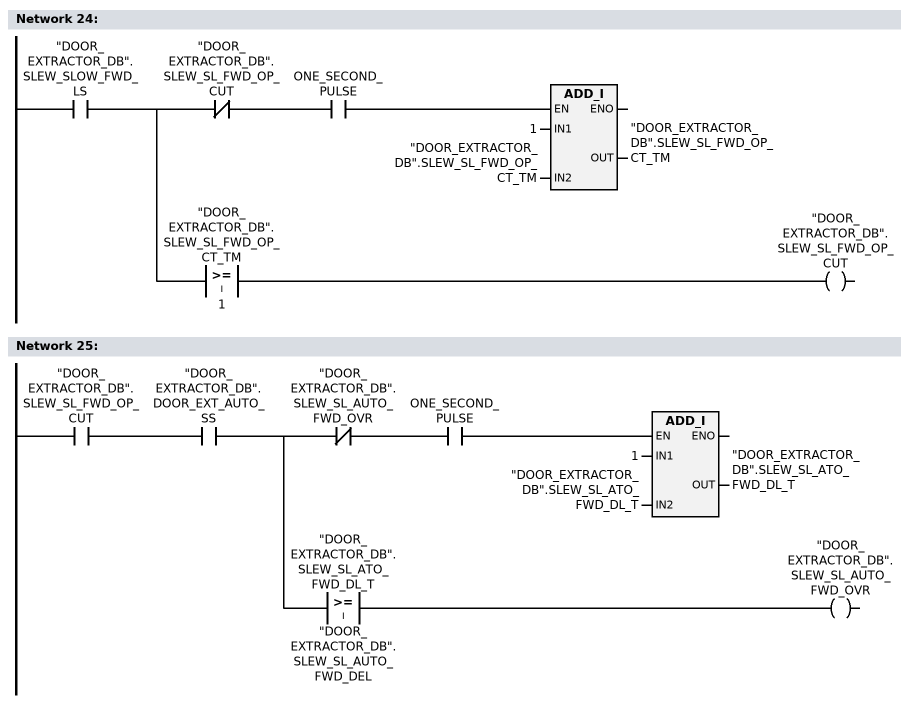
NETWORK
TITLE =
      A     "DOOR_EXTRACTOR_DB".SLEW_SLOW_FWD_LS;
      =     L 0.0;
      A     L 0.0;
      AN    "DOOR_EXTRACTOR_DB".SLEW_SL_FWD_OP_CUT;
      A     "ONE_SECOND_PULSE";
      JNB   _011;
      L     1;
      L     "DOOR_EXTRACTOR_DB".SLEW_SL_FWD_OP_CT_TM;
      +I;
      T     "DOOR_EXTRACTOR_DB".SLEW_SL_FWD_OP_CT_TM;
_011: NOP   0;
      A     L 0.0;
      A(;
      L     "DOOR_EXTRACTOR_DB".SLEW_SL_FWD_OP_CT_TM;
      L     1;
      >=I;
      );
      =     "DOOR_EXTRACTOR_DB".SLEW_SL_FWD_OP_CUT;
NETWORK
TITLE =
      A     "DOOR_EXTRACTOR_DB".SLEW_SL_FWD_OP_CUT;
      A     "DOOR_EXTRACTOR_DB".DOOR_EXT_AUTO_SS;
      =     L 0.0;
      A     L 0.0;
      AN    "DOOR_EXTRACTOR_DB".SLEW_SL_AUTO_FWD_OVR;
      A     "ONE_SECOND_PULSE";
      JNB   _012;
      L     1;
      L     "DOOR_EXTRACTOR_DB".SLEW_SL_ATO_FWD_DL_T;
      +I;
      T     "DOOR_EXTRACTOR_DB".SLEW_SL_ATO_FWD_DL_T;
_012: NOP   0;
      A     L 0.0;
      A(;
      L     "DOOR_EXTRACTOR_DB".SLEW_SL_ATO_FWD_DL_T;
      L     "DOOR_EXTRACTOR_DB".SLEW_SL_AUTO_FWD_DEL;
      >=I;
      );
      =     "DOOR_EXTRACTOR_DB".SLEW_SL_AUTO_FWD_OVR;
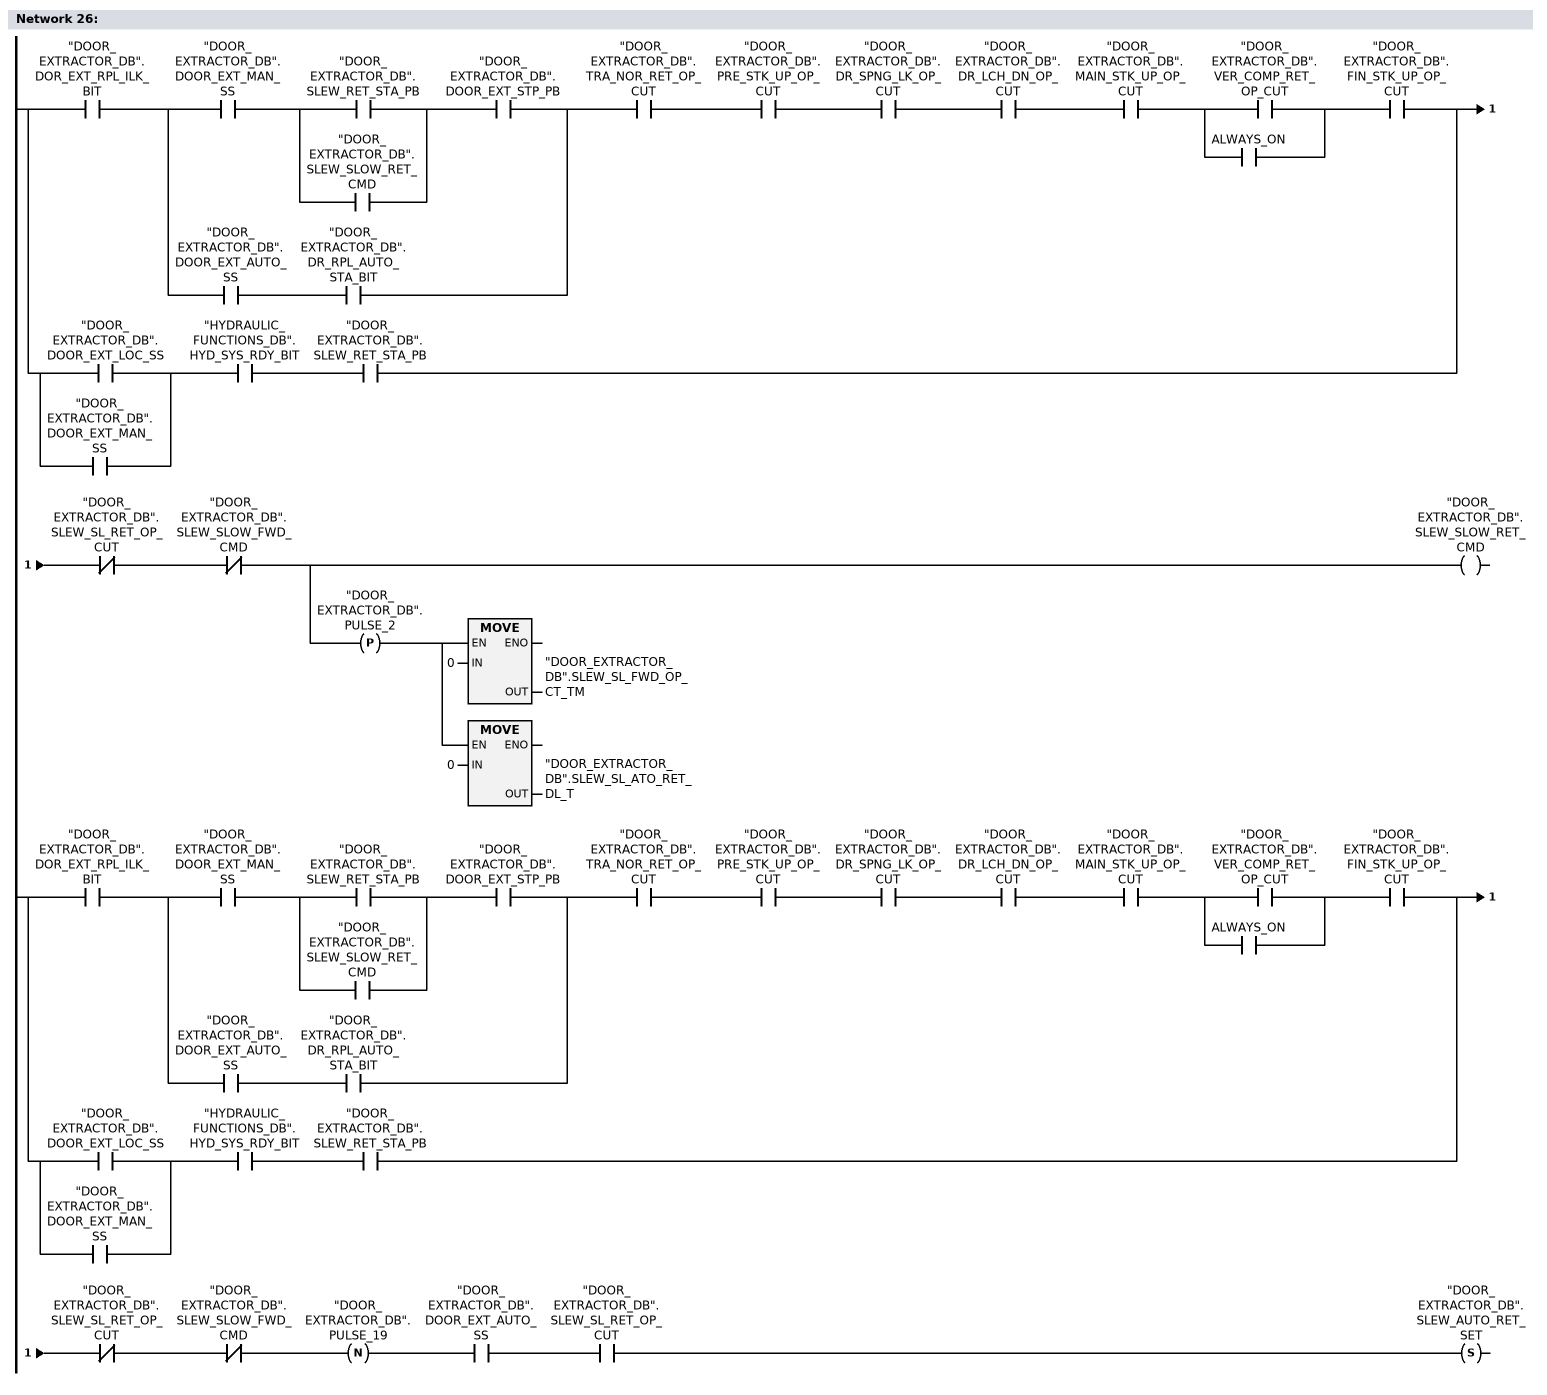
NETWORK
TITLE =
      A(;
      A     "DOOR_EXTRACTOR_DB".DOR_EXT_RPL_ILK_BIT;
      A(;
      A     "DOOR_EXTRACTOR_DB".DOOR_EXT_MAN_SS;
      A(;
      O     "DOOR_EXTRACTOR_DB".SLEW_RET_STA_PB;
      O     "DOOR_EXTRACTOR_DB".SLEW_SLOW_RET_CMD;
      );
      A     "DOOR_EXTRACTOR_DB".DOOR_EXT_STP_PB;
      O;
      A     "DOOR_EXTRACTOR_DB".DOOR_EXT_AUTO_SS;
      A     "DOOR_EXTRACTOR_DB".DR_RPL_AUTO_STA_BIT;
      );
      A     "DOOR_EXTRACTOR_DB".TRA_NOR_RET_OP_CUT;
      A     "DOOR_EXTRACTOR_DB".PRE_STK_UP_OP_CUT;
      A     "DOOR_EXTRACTOR_DB".DR_SPNG_LK_OP_CUT;
      A     "DOOR_EXTRACTOR_DB".DR_LCH_DN_OP_CUT;
      A     "DOOR_EXTRACTOR_DB".MAIN_STK_UP_OP_CUT;
      A(;
      O     "DOOR_EXTRACTOR_DB".VER_COMP_RET_OP_CUT;
      O     "ALWAYS_ON";
      );
      A     "DOOR_EXTRACTOR_DB".FIN_STK_UP_OP_CUT;
      O;
      A(;
      O     "DOOR_EXTRACTOR_DB".DOOR_EXT_LOC_SS;
      O     "DOOR_EXTRACTOR_DB".DOOR_EXT_MAN_SS;
      );
      A     "HYDRAULIC_FUNCTIONS_DB".HYD_SYS_RDY_BIT;
      A     "DOOR_EXTRACTOR_DB".SLEW_RET_STA_PB;
      );
      AN    "DOOR_EXTRACTOR_DB".SLEW_SL_RET_OP_CUT;
      AN    "DOOR_EXTRACTOR_DB".SLEW_SLOW_FWD_CMD;
      =     L 0.0;
      A     L 0.0;
      BLD   102;
      =     "DOOR_EXTRACTOR_DB".SLEW_SLOW_RET_CMD;
      A(;
      A     L 0.0;
      FN    "DOOR_EXTRACTOR_DB".PULSE_19;
      );
      A     "DOOR_EXTRACTOR_DB".DOOR_EXT_AUTO_SS;
      A     "DOOR_EXTRACTOR_DB".SLEW_SL_RET_OP_CUT;
      S     "DOOR_EXTRACTOR_DB".SLEW_AUTO_RET_SET;
      A     L 0.0;
      FP    "DOOR_EXTRACTOR_DB".PULSE_2;
      =     L 0.1;
      A     L 0.1;
      JNB   _013;
      L     0;
      T     "DOOR_EXTRACTOR_DB".SLEW_SL_FWD_OP_CT_TM;
_013: NOP   0;
      A     L 0.1;
      JNB   _014;
      L     0;
      T     "DOOR_EXTRACTOR_DB".SLEW_SL_ATO_RET_DL_T;
_014: NOP   0;
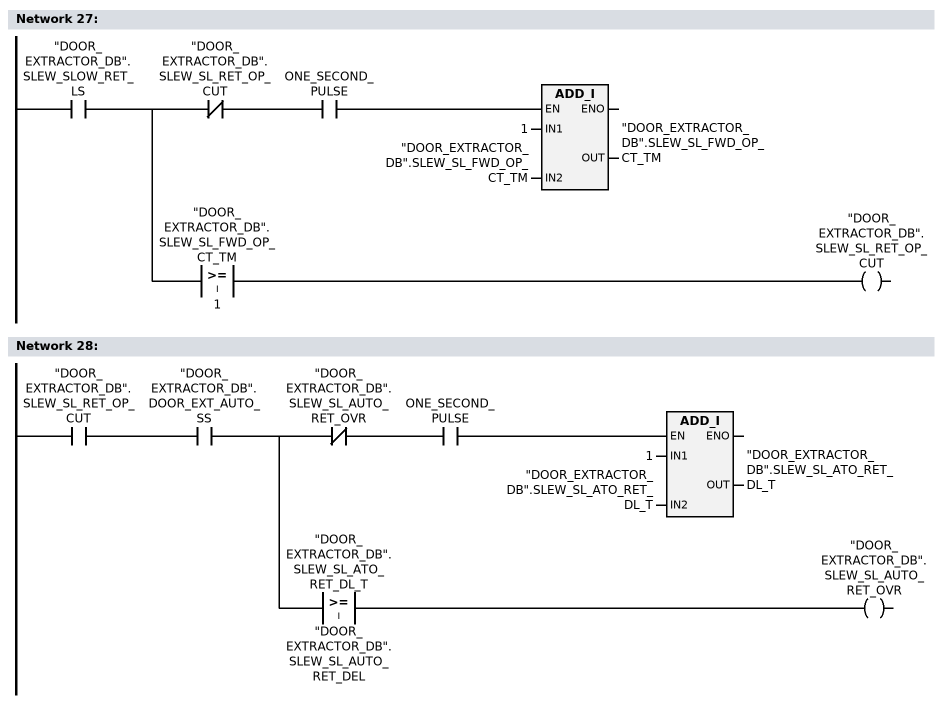
NETWORK
TITLE =
      A     "DOOR_EXTRACTOR_DB".SLEW_SLOW_RET_LS;
      =     L 0.0;
      A     L 0.0;
      AN    "DOOR_EXTRACTOR_DB".SLEW_SL_RET_OP_CUT;
      A     "ONE_SECOND_PULSE";
      JNB   _015;
      L     1;
      L     "DOOR_EXTRACTOR_DB".SLEW_SL_FWD_OP_CT_TM;
      +I;
      T     "DOOR_EXTRACTOR_DB".SLEW_SL_FWD_OP_CT_TM;
_015: NOP   0;
      A     L 0.0;
      A(;
      L     "DOOR_EXTRACTOR_DB".SLEW_SL_FWD_OP_CT_TM;
      L     1;
      >=I;
      );
      =     "DOOR_EXTRACTOR_DB".SLEW_SL_RET_OP_CUT;
NETWORK
TITLE =
      A     "DOOR_EXTRACTOR_DB".SLEW_SL_RET_OP_CUT;
      A     "DOOR_EXTRACTOR_DB".DOOR_EXT_AUTO_SS;
      =     L 0.0;
      A     L 0.0;
      AN    "DOOR_EXTRACTOR_DB".SLEW_SL_AUTO_RET_OVR;
      A     "ONE_SECOND_PULSE";
      JNB   _016;
      L     1;
      L     "DOOR_EXTRACTOR_DB".SLEW_SL_ATO_RET_DL_T;
      +I;
      T     "DOOR_EXTRACTOR_DB".SLEW_SL_ATO_RET_DL_T;
_016: NOP   0;
      A     L 0.0;
      A(;
      L     "DOOR_EXTRACTOR_DB".SLEW_SL_ATO_RET_DL_T;
      L     "DOOR_EXTRACTOR_DB".SLEW_SL_AUTO_RET_DEL;
      >=I;
      );
      =     "DOOR_EXTRACTOR_DB".SLEW_SL_AUTO_RET_OVR;
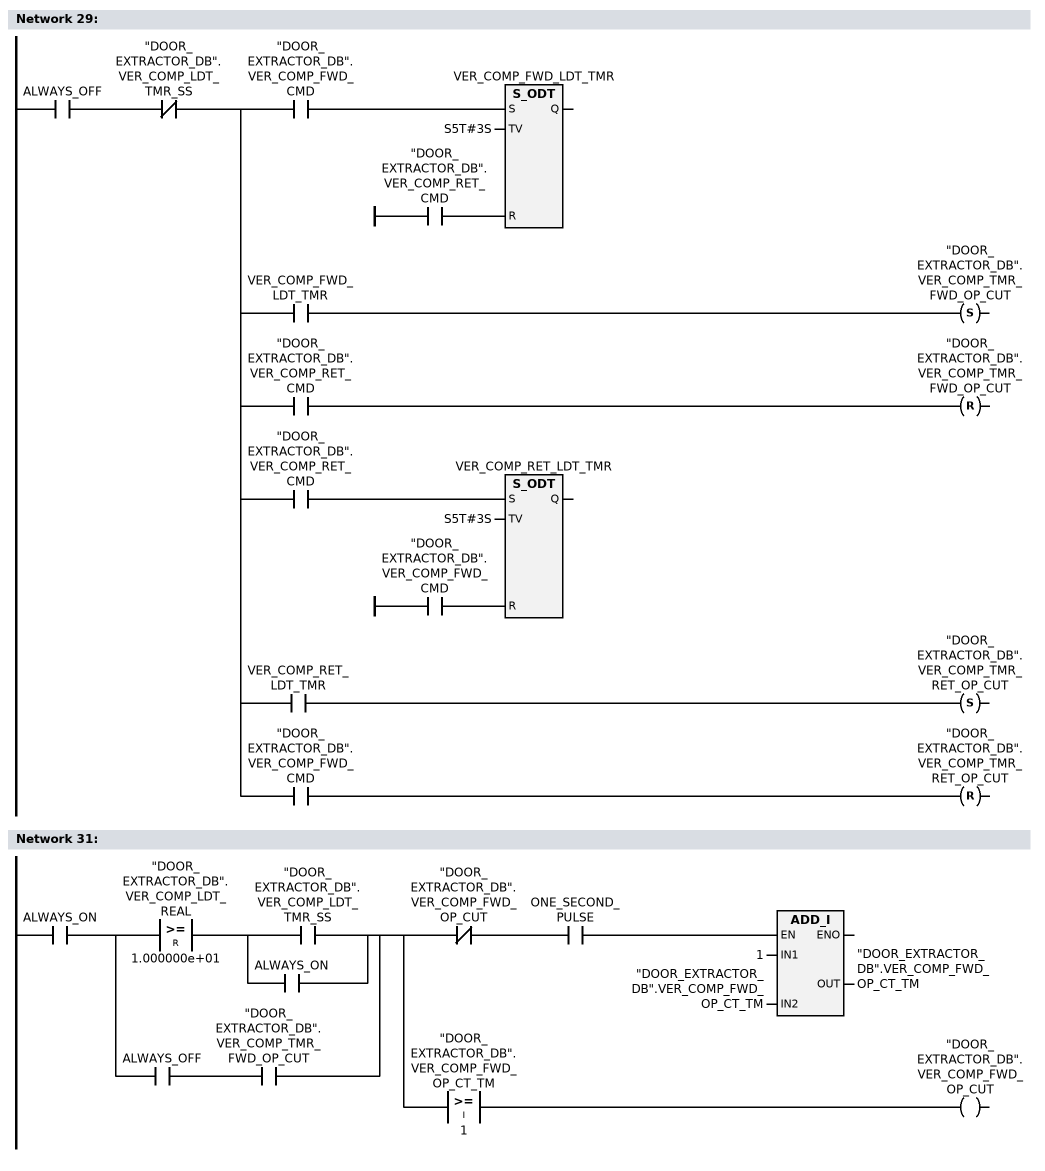
NETWORK
TITLE =
      A     "ALWAYS_OFF";
      AN    "DOOR_EXTRACTOR_DB".VER_COMP_LDT_TMR_SS;
      =     L 0.0;
      A     L 0.0;
      A     "DOOR_EXTRACTOR_DB".VER_COMP_FWD_CMD;
      L     S5T#3S;
      SD    "VER_COMP_FWD_LDT_TMR";
      A     "DOOR_EXTRACTOR_DB".VER_COMP_RET_CMD;
      R     "VER_COMP_FWD_LDT_TMR";
      NOP   0;
      NOP   0;
      NOP   0;
      A     L 0.0;
      A     "VER_COMP_FWD_LDT_TMR";
      S     "DOOR_EXTRACTOR_DB".VER_COMP_TMR_FWD_OP_CUT;
      A     L 0.0;
      A     "DOOR_EXTRACTOR_DB".VER_COMP_RET_CMD;
      R     "DOOR_EXTRACTOR_DB".VER_COMP_TMR_FWD_OP_CUT;
      A     L 0.0;
      A     "DOOR_EXTRACTOR_DB".VER_COMP_RET_CMD;
      L     S5T#3S;
      SD    "VER_COMP_RET_LDT_TMR";
      A     "DOOR_EXTRACTOR_DB".VER_COMP_FWD_CMD;
      R     "VER_COMP_RET_LDT_TMR";
      NOP   0;
      NOP   0;
      NOP   0;
      A     L 0.0;
      A     "VER_COMP_RET_LDT_TMR";
      S     "DOOR_EXTRACTOR_DB".VER_COMP_TMR_RET_OP_CUT;
      A     L 0.0;
      A     "DOOR_EXTRACTOR_DB".VER_COMP_FWD_CMD;
      R     "DOOR_EXTRACTOR_DB".VER_COMP_TMR_RET_OP_CUT;
NETWORK
TITLE =
      A(;
      A     "DOOR_EXTRACTOR_DB".DOR_EXT_RPL_ILK_BIT;
      A(;
      A     "DOOR_EXTRACTOR_DB".DOOR_EXT_MAN_SS;
      A(;
      O     "DOOR_EXTRACTOR_DB".VER_COMP_FWD_STA_PB;
      O     "DOOR_EXTRACTOR_DB".VER_COMP_FWD_CMD;
      );
      A     "DOOR_EXTRACTOR_DB".DOOR_EXT_STP_PB;
      O;
      A     "DOOR_EXTRACTOR_DB".DOOR_EXT_AUTO_SS;
      A(;
      A     "DOOR_EXTRACTOR_DB".DR_EXT_AUTO_STA_BIT;
      A(;
      ON    "DOOR_EXTRACTOR_DB".VER_COMP_AUTO_FWD_SET;
      O     "ALWAYS_ON";
      );
      O;
      A     "DOOR_EXTRACTOR_DB".DR_RPL_AUTO_STA_BIT;
      A     "DOOR_EXTRACTOR_DB".FIN_STK_AUTO_RET_SET;
      A(;
      ON    "DOOR_EXTRACTOR_DB".VER_COMP_AUTO_FWD_SET;
      O     "ALWAYS_ON";
      );
      );
      );
      A(;
      A     "DOOR_EXTRACTOR_DB".SLEW_NR_RET_OP_CUT;
      A     "DOOR_EXTRACTOR_DB".PRE_STK_DN_OP_CUT;
      A     "DOOR_EXTRACTOR_DB".MAIN_STK_DN_OP_CUT;
      A     "DOOR_EXTRACTOR_DB".DR_LCH_UP_OP_CUT;
      A     "DOOR_EXTRACTOR_DB".DR_SPNG_UNLK_OP_CUT;
      O;
      A     "DOOR_EXTRACTOR_DB".SLEW_NR_RET_OP_CUT;
      A     "DOOR_EXTRACTOR_DB".TRA_NOR_RET_OP_CUT;
      A     "DOOR_EXTRACTOR_DB".PRE_STK_UP_OP_CUT;
      A     "DOOR_EXTRACTOR_DB".DR_SPNG_LK_OP_CUT;
      A     "DOOR_EXTRACTOR_DB".DR_LCH_DN_OP_CUT;
      A     "DOOR_EXTRACTOR_DB".MAIN_STK_UP_OP_CUT;
      A     "DOOR_EXTRACTOR_DB".FIN_STK_DN_OP_CUT;
      );
      O;
      A(;
      O     "DOOR_EXTRACTOR_DB".DOOR_EXT_LOC_SS;
      O     "DOOR_EXTRACTOR_DB".DOOR_EXT_MAN_SS;
      );
      A     "HYDRAULIC_FUNCTIONS_DB".HYD_SYS_RDY_BIT;
      A     "DOOR_EXTRACTOR_DB".VER_COMP_FWD_STA_PB;
      );
      AN    "DOOR_EXTRACTOR_DB".VER_COMP_FWD_OP_CUT;
      AN    "DOOR_EXTRACTOR_DB".VER_COMP_RET_CMD;
      =     L 0.0;
      A     L 0.0;
      AN    "DOOR_EXTRACTOR_DB".DOOR_EXT_AUTO_SS;
      =     L 0.1;
      A     L 0.1;
      BLD   102;
      =     "DOOR_EXTRACTOR_DB".VER_COMP_FWD_CMD;
      A(;
      A     L 0.1;
      FN    "DOOR_EXTRACTOR_DB".PULSE_20;
      );
      A     "DOOR_EXTRACTOR_DB".VER_COMP_FWD_OP_CUT;
      A     "DOOR_EXTRACTOR_DB".DOOR_EXT_AUTO_SS;
      S     "DOOR_EXTRACTOR_DB".VER_COMP_AUTO_FWD_SET;
      A     L 0.0;
      FP    "DOOR_EXTRACTOR_DB".PULSE_3;
      =     L 0.1;
      A     L 0.1;
      A     "DOOR_EXTRACTOR_DB".DOOR_EXT_AUTO_SS;
      S     "DOOR_EXTRACTOR_DB".VER_COMP_AUTO_FWD_SET;
      A     L 0.1;
      JNB   _017;
      L     0;
      T     "DOOR_EXTRACTOR_DB".VER_COMP_FWD_OP_CT_TM;
_017: NOP   0;
      A     L 0.1;
      JNB   _018;
      L     0;
      T     "DOOR_EXTRACTOR_DB".VER_COMP_ATO_FWD_DL_T;
_018: NOP   0;
NETWORK
TITLE =
      A     "ALWAYS_ON";
      A(;
      A(;
      L     "DOOR_EXTRACTOR_DB".VER_COMP_LDT_REAL;
      L     1.000000e+01;
      >=R;
      );
      A(;
      O     "DOOR_EXTRACTOR_DB".VER_COMP_LDT_TMR_SS;
      O     "ALWAYS_ON";
      );
      O;
      A     "ALWAYS_OFF";
      A     "DOOR_EXTRACTOR_DB".VER_COMP_TMR_FWD_OP_CUT;
      );
      =     L 0.0;
      A     L 0.0;
      AN    "DOOR_EXTRACTOR_DB".VER_COMP_FWD_OP_CUT;
      A     "ONE_SECOND_PULSE";
      JNB   _019;
      L     1;
      L     "DOOR_EXTRACTOR_DB".VER_COMP_FWD_OP_CT_TM;
      +I;
      T     "DOOR_EXTRACTOR_DB".VER_COMP_FWD_OP_CT_TM;
_019: NOP   0;
      A     L 0.0;
      A(;
      L     "DOOR_EXTRACTOR_DB".VER_COMP_FWD_OP_CT_TM;
      L     1;
      >=I;
      );
      =     "DOOR_EXTRACTOR_DB".VER_COMP_FWD_OP_CUT;
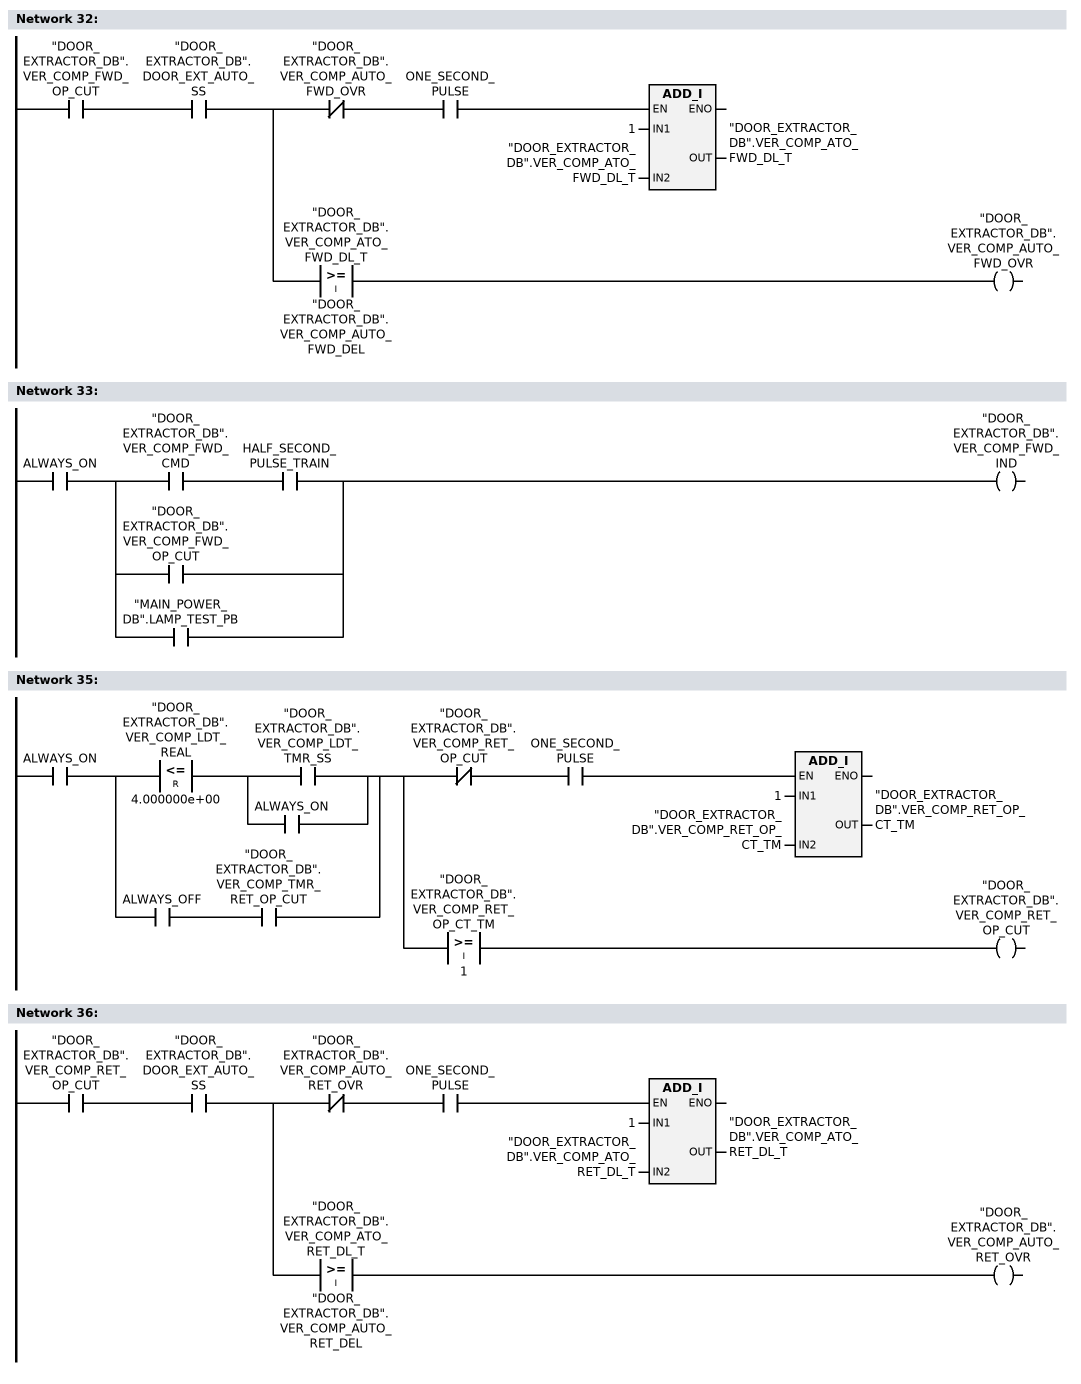
NETWORK
TITLE =
      A     "DOOR_EXTRACTOR_DB".VER_COMP_FWD_OP_CUT;
      A     "DOOR_EXTRACTOR_DB".DOOR_EXT_AUTO_SS;
      =     L 0.0;
      A     L 0.0;
      AN    "DOOR_EXTRACTOR_DB".VER_COMP_AUTO_FWD_OVR;
      A     "ONE_SECOND_PULSE";
      JNB   _01a;
      L     1;
      L     "DOOR_EXTRACTOR_DB".VER_COMP_ATO_FWD_DL_T;
      +I;
      T     "DOOR_EXTRACTOR_DB".VER_COMP_ATO_FWD_DL_T;
_01a: NOP   0;
      A     L 0.0;
      A(;
      L     "DOOR_EXTRACTOR_DB".VER_COMP_ATO_FWD_DL_T;
      L     "DOOR_EXTRACTOR_DB".VER_COMP_AUTO_FWD_DEL;
      >=I;
      );
      =     "DOOR_EXTRACTOR_DB".VER_COMP_AUTO_FWD_OVR;
NETWORK
TITLE =
      A     "ALWAYS_ON";
      A(;
      A     "DOOR_EXTRACTOR_DB".VER_COMP_FWD_CMD;
      A     "HALF_SECOND_PULSE_TRAIN";
      O     "DOOR_EXTRACTOR_DB".VER_COMP_FWD_OP_CUT;
      O     "MAIN_POWER_DB".LAMP_TEST_PB;
      );
      =     "DOOR_EXTRACTOR_DB".VER_COMP_FWD_IND;
NETWORK
TITLE =
      A(;
      A     "DOOR_EXTRACTOR_DB".DOR_EXT_RPL_ILK_BIT;
      A(;
      A     "DOOR_EXTRACTOR_DB".DOOR_EXT_MAN_SS;
      A(;
      O     "DOOR_EXTRACTOR_DB".VER_COMP_RET_STA_PB;
      O     "DOOR_EXTRACTOR_DB".VER_COMP_RET_CMD;
      );
      A     "DOOR_EXTRACTOR_DB".DOOR_EXT_STP_PB;
      O;
      A     "DOOR_EXTRACTOR_DB".DOOR_EXT_AUTO_SS;
      A(;
      A     "DOOR_EXTRACTOR_DB".DR_EXT_AUTO_STA_BIT;
      A     "DOOR_EXTRACTOR_DB".TRA_AUTO_RET_SET;
      A     "DOOR_EXTRACTOR_DB".TRA_NOR_AUTO_RET_OVR;
      O;
      A     "DOOR_EXTRACTOR_DB".DR_RPL_AUTO_STA_BIT;
      A     "DOOR_EXTRACTOR_DB".TRA_AUTO_RET_SET;
      A     "DOOR_EXTRACTOR_DB".TRA_NOR_AUTO_RET_OVR;
      );
      );
      A(;
      A     "DOOR_EXTRACTOR_DB".SLEW_NR_RET_OP_CUT;
      A     "DOOR_EXTRACTOR_DB".TRA_NOR_RET_OP_CUT;
      A     "DOOR_EXTRACTOR_DB".PRE_STK_UP_OP_CUT;
      A     "DOOR_EXTRACTOR_DB".DR_SPNG_LK_OP_CUT;
      A     "DOOR_EXTRACTOR_DB".DR_LCH_DN_OP_CUT;
      A     "DOOR_EXTRACTOR_DB".MAIN_STK_UP_OP_CUT;
      O;
      A     "DOOR_EXTRACTOR_DB".SLEW_NR_RET_OP_CUT;
      A     "DOOR_EXTRACTOR_DB".TRA_NOR_RET_OP_CUT;
      A     "DOOR_EXTRACTOR_DB".PRE_STK_DN_OP_CUT;
      A     "DOOR_EXTRACTOR_DB".DR_SPNG_UNLK_OP_CUT;
      A     "DOOR_EXTRACTOR_DB".DR_LCH_UP_OP_CUT;
      A     "DOOR_EXTRACTOR_DB".MAIN_STK_DN_OP_CUT;
      A     "DOOR_EXTRACTOR_DB".FIN_STK_DN_OP_CUT;
      );
      O;
      A(;
      O     "DOOR_EXTRACTOR_DB".DOOR_EXT_LOC_SS;
      O     "DOOR_EXTRACTOR_DB".DOOR_EXT_MAN_SS;
      );
      A     "HYDRAULIC_FUNCTIONS_DB".HYD_SYS_RDY_BIT;
      A     "DOOR_EXTRACTOR_DB".VER_COMP_RET_STA_PB;
      );
      AN    "DOOR_EXTRACTOR_DB".VER_COMP_RET_OP_CUT;
      AN    "DOOR_EXTRACTOR_DB".VER_COMP_FWD_CMD;
      =     L 0.0;
      A     L 0.0;
      AN    "DOOR_EXTRACTOR_DB".DOOR_EXT_AUTO_SS;
      =     L 0.1;
      A     L 0.1;
      BLD   102;
      =     "DOOR_EXTRACTOR_DB".VER_COMP_RET_CMD;
      A(;
      A     L 0.1;
      FN    "DOOR_EXTRACTOR_DB".PULSE_21;
      );
      A     "DOOR_EXTRACTOR_DB".DOOR_EXT_AUTO_SS;
      A     "DOOR_EXTRACTOR_DB".VER_COMP_RET_OP_CUT;
      S     "DOOR_EXTRACTOR_DB".VER_COMP_AUTO_RET_SET;
      A     L 0.0;
      FP    "DOOR_EXTRACTOR_DB".PULSE_4;
      =     L 0.1;
      A     L 0.1;
      A     "DOOR_EXTRACTOR_DB".DOOR_EXT_AUTO_SS;
      S     "DOOR_EXTRACTOR_DB".VER_COMP_AUTO_RET_SET;
      A     L 0.1;
      JNB   _01b;
      L     0;
      T     "DOOR_EXTRACTOR_DB".VER_COMP_RET_OP_CT_TM;
_01b: NOP   0;
      A     L 0.1;
      JNB   _01c;
      L     0;
      T     "DOOR_EXTRACTOR_DB".VER_COMP_ATO_RET_DL_T;
_01c: NOP   0;
NETWORK
TITLE =
      A     "ALWAYS_ON";
      A(;
      A(;
      L     "DOOR_EXTRACTOR_DB".VER_COMP_LDT_REAL;
      L     4.000000e+00;
      <=R;
      );
      A(;
      O     "DOOR_EXTRACTOR_DB".VER_COMP_LDT_TMR_SS;
      O     "ALWAYS_ON";
      );
      O;
      A     "ALWAYS_OFF";
      A     "DOOR_EXTRACTOR_DB".VER_COMP_TMR_RET_OP_CUT;
      );
      =     L 0.0;
      A     L 0.0;
      AN    "DOOR_EXTRACTOR_DB".VER_COMP_RET_OP_CUT;
      A     "ONE_SECOND_PULSE";
      JNB   _01d;
      L     1;
      L     "DOOR_EXTRACTOR_DB".VER_COMP_RET_OP_CT_TM;
      +I;
      T     "DOOR_EXTRACTOR_DB".VER_COMP_RET_OP_CT_TM;
_01d: NOP   0;
      A     L 0.0;
      A(;
      L     "DOOR_EXTRACTOR_DB".VER_COMP_RET_OP_CT_TM;
      L     1;
      >=I;
      );
      =     "DOOR_EXTRACTOR_DB".VER_COMP_RET_OP_CUT;
NETWORK
TITLE =
      A     "DOOR_EXTRACTOR_DB".VER_COMP_RET_OP_CUT;
      A     "DOOR_EXTRACTOR_DB".DOOR_EXT_AUTO_SS;
      =     L 0.0;
      A     L 0.0;
      AN    "DOOR_EXTRACTOR_DB".VER_COMP_AUTO_RET_OVR;
      A     "ONE_SECOND_PULSE";
      JNB   _01e;
      L     1;
      L     "DOOR_EXTRACTOR_DB".VER_COMP_ATO_RET_DL_T;
      +I;
      T     "DOOR_EXTRACTOR_DB".VER_COMP_ATO_RET_DL_T;
_01e: NOP   0;
      A     L 0.0;
      A(;
      L     "DOOR_EXTRACTOR_DB".VER_COMP_ATO_RET_DL_T;
      L     "DOOR_EXTRACTOR_DB".VER_COMP_AUTO_RET_DEL;
      >=I;
      );
      =     "DOOR_EXTRACTOR_DB".VER_COMP_AUTO_RET_OVR;
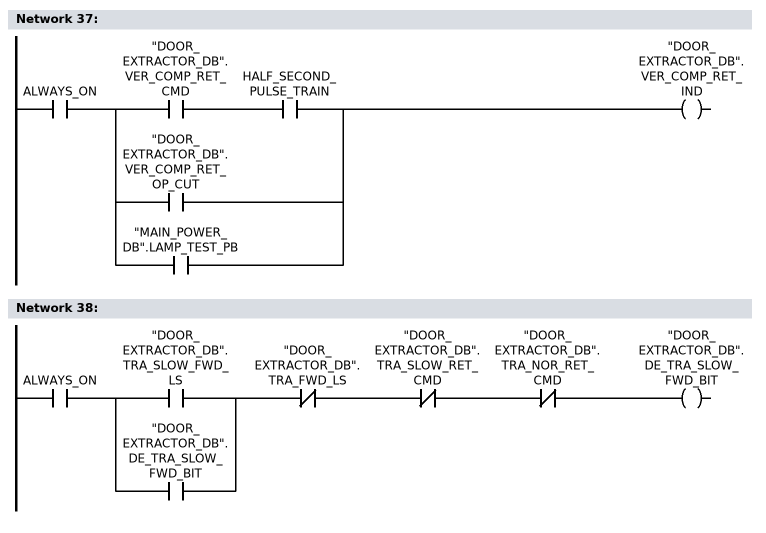
NETWORK
TITLE =
      A     "ALWAYS_ON";
      A(;
      A     "DOOR_EXTRACTOR_DB".VER_COMP_RET_CMD;
      A     "HALF_SECOND_PULSE_TRAIN";
      O     "DOOR_EXTRACTOR_DB".VER_COMP_RET_OP_CUT;
      O     "MAIN_POWER_DB".LAMP_TEST_PB;
      );
      =     "DOOR_EXTRACTOR_DB".VER_COMP_RET_IND;
NETWORK
TITLE =
      A     "ALWAYS_ON";
      A(;
      O     "DOOR_EXTRACTOR_DB".TRA_SLOW_FWD_LS;
      O     "DOOR_EXTRACTOR_DB".DE_TRA_SLOW_FWD_BIT;
      );
      AN    "DOOR_EXTRACTOR_DB".TRA_FWD_LS;
      AN    "DOOR_EXTRACTOR_DB".TRA_SLOW_RET_CMD;
      AN    "DOOR_EXTRACTOR_DB".TRA_NOR_RET_CMD;
      =     "DOOR_EXTRACTOR_DB".DE_TRA_SLOW_FWD_BIT;
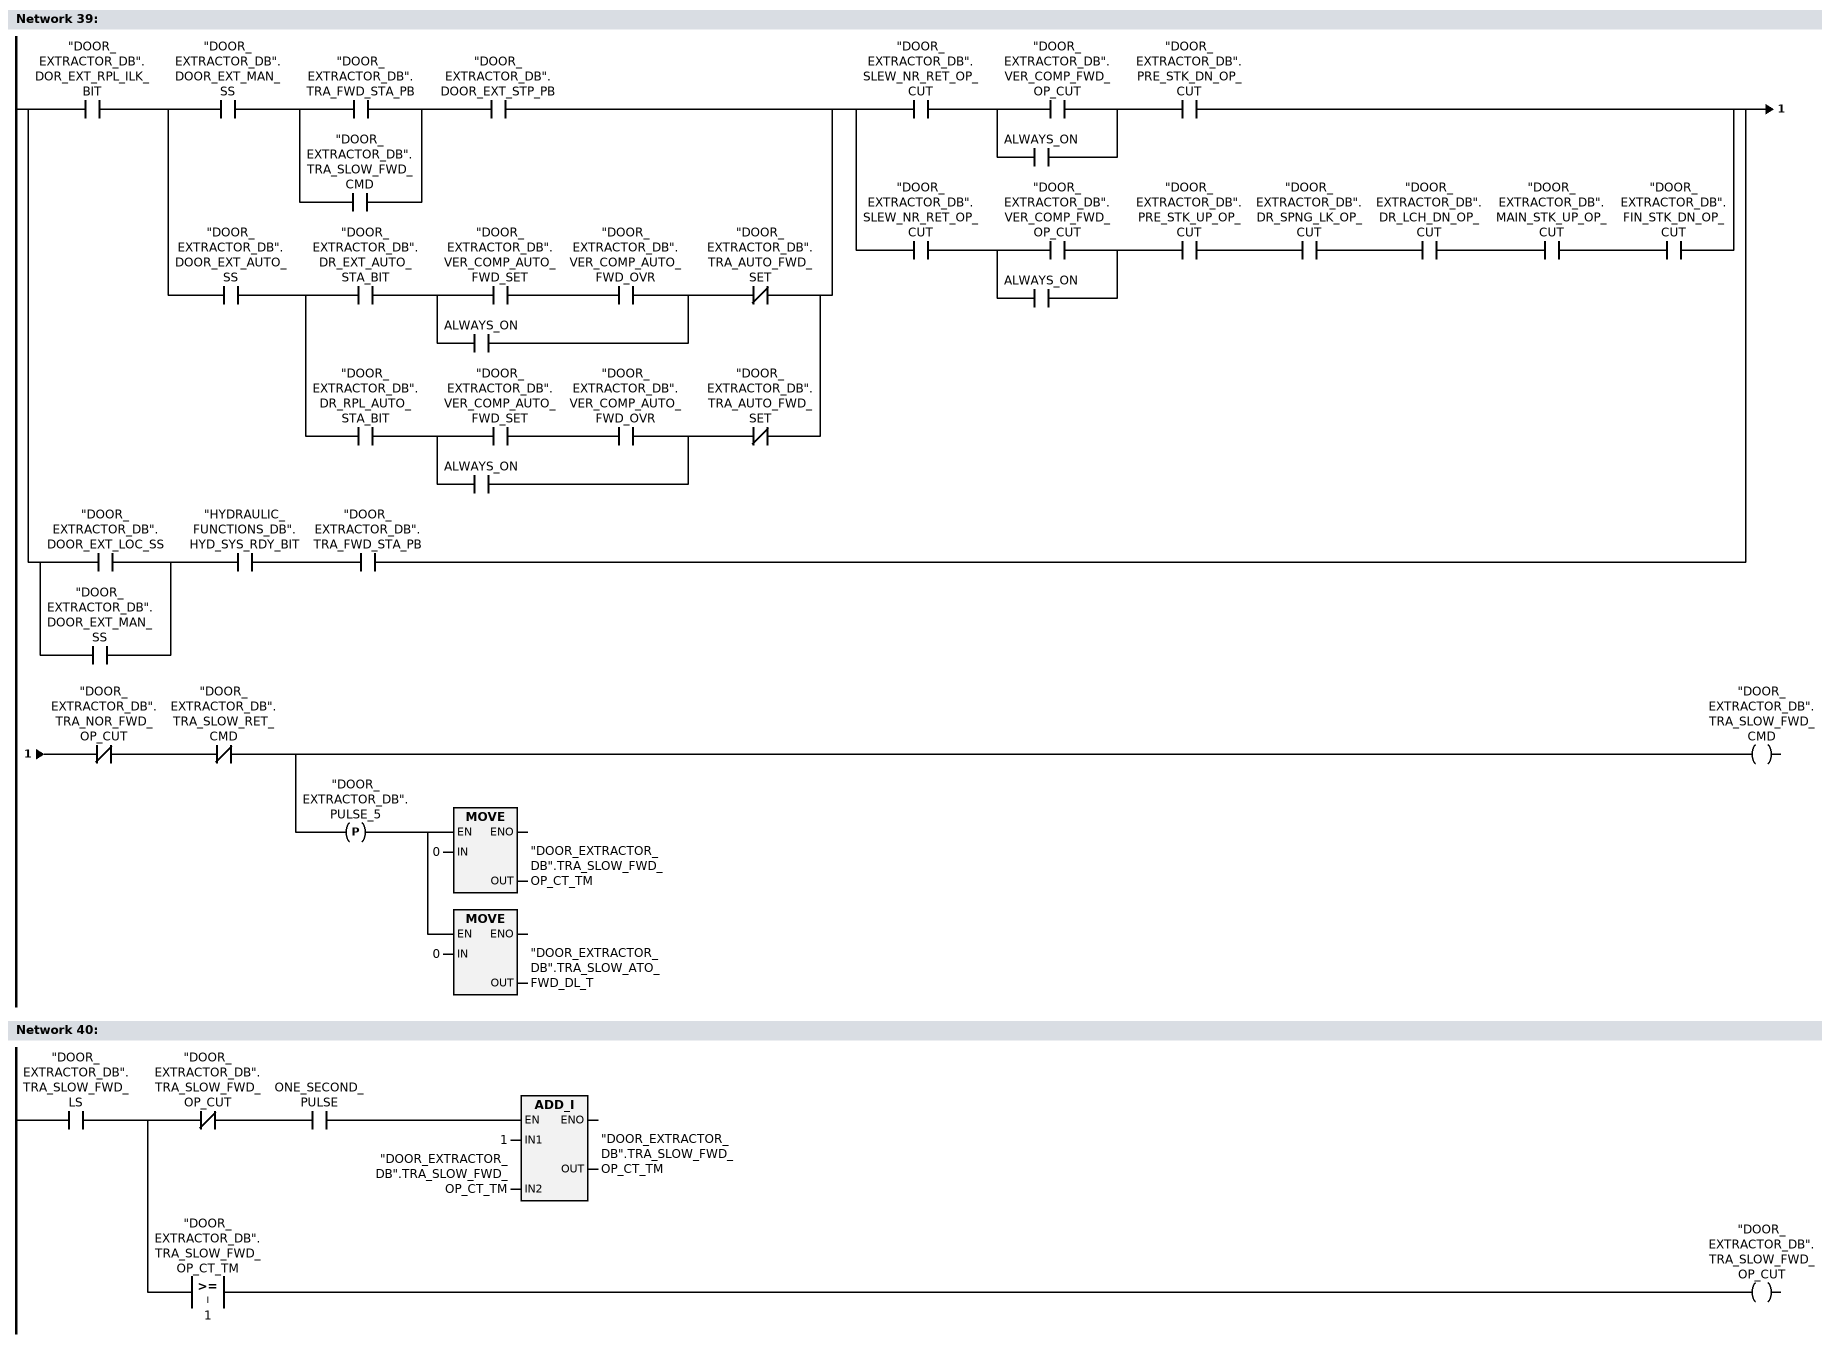
NETWORK
TITLE =
      A(;
      A     "DOOR_EXTRACTOR_DB".DOR_EXT_RPL_ILK_BIT;
      A(;
      A     "DOOR_EXTRACTOR_DB".DOOR_EXT_MAN_SS;
      A(;
      O     "DOOR_EXTRACTOR_DB".TRA_FWD_STA_PB;
      O     "DOOR_EXTRACTOR_DB".TRA_SLOW_FWD_CMD;
      );
      A     "DOOR_EXTRACTOR_DB".DOOR_EXT_STP_PB;
      O;
      A     "DOOR_EXTRACTOR_DB".DOOR_EXT_AUTO_SS;
      A(;
      A     "DOOR_EXTRACTOR_DB".DR_EXT_AUTO_STA_BIT;
      A(;
      A     "DOOR_EXTRACTOR_DB".VER_COMP_AUTO_FWD_SET;
      A     "DOOR_EXTRACTOR_DB".VER_COMP_AUTO_FWD_OVR;
      O     "ALWAYS_ON";
      );
      AN    "DOOR_EXTRACTOR_DB".TRA_AUTO_FWD_SET;
      O;
      A     "DOOR_EXTRACTOR_DB".DR_RPL_AUTO_STA_BIT;
      A(;
      A     "DOOR_EXTRACTOR_DB".VER_COMP_AUTO_FWD_SET;
      A     "DOOR_EXTRACTOR_DB".VER_COMP_AUTO_FWD_OVR;
      O     "ALWAYS_ON";
      );
      AN    "DOOR_EXTRACTOR_DB".TRA_AUTO_FWD_SET;
      );
      );
      A(;
      A     "DOOR_EXTRACTOR_DB".SLEW_NR_RET_OP_CUT;
      A(;
      O     "DOOR_EXTRACTOR_DB".VER_COMP_FWD_OP_CUT;
      O     "ALWAYS_ON";
      );
      A     "DOOR_EXTRACTOR_DB".PRE_STK_DN_OP_CUT;
      O;
      A     "DOOR_EXTRACTOR_DB".SLEW_NR_RET_OP_CUT;
      A(;
      O     "DOOR_EXTRACTOR_DB".VER_COMP_FWD_OP_CUT;
      O     "ALWAYS_ON";
      );
      A     "DOOR_EXTRACTOR_DB".PRE_STK_UP_OP_CUT;
      A     "DOOR_EXTRACTOR_DB".DR_SPNG_LK_OP_CUT;
      A     "DOOR_EXTRACTOR_DB".DR_LCH_DN_OP_CUT;
      A     "DOOR_EXTRACTOR_DB".MAIN_STK_UP_OP_CUT;
      A     "DOOR_EXTRACTOR_DB".FIN_STK_DN_OP_CUT;
      );
      O;
      A(;
      O     "DOOR_EXTRACTOR_DB".DOOR_EXT_LOC_SS;
      O     "DOOR_EXTRACTOR_DB".DOOR_EXT_MAN_SS;
      );
      A     "HYDRAULIC_FUNCTIONS_DB".HYD_SYS_RDY_BIT;
      A     "DOOR_EXTRACTOR_DB".TRA_FWD_STA_PB;
      );
      AN    "DOOR_EXTRACTOR_DB".TRA_NOR_FWD_OP_CUT;
      AN    "DOOR_EXTRACTOR_DB".TRA_SLOW_RET_CMD;
      =     L 0.0;
      A     L 0.0;
      BLD   102;
      =     "DOOR_EXTRACTOR_DB".TRA_SLOW_FWD_CMD;
      A     L 0.0;
      FP    "DOOR_EXTRACTOR_DB".PULSE_5;
      =     L 0.1;
      A     L 0.1;
      JNB   _01f;
      L     0;
      T     "DOOR_EXTRACTOR_DB".TRA_SLOW_FWD_OP_CT_TM;
_01f: NOP   0;
      A     L 0.1;
      JNB   _020;
      L     0;
      T     "DOOR_EXTRACTOR_DB".TRA_SLOW_ATO_FWD_DL_T;
_020: NOP   0;
NETWORK
TITLE =
      A     "DOOR_EXTRACTOR_DB".TRA_SLOW_FWD_LS;
      =     L 0.0;
      A     L 0.0;
      AN    "DOOR_EXTRACTOR_DB".TRA_SLOW_FWD_OP_CUT;
      A     "ONE_SECOND_PULSE";
      JNB   _021;
      L     1;
      L     "DOOR_EXTRACTOR_DB".TRA_SLOW_FWD_OP_CT_TM;
      +I;
      T     "DOOR_EXTRACTOR_DB".TRA_SLOW_FWD_OP_CT_TM;
_021: NOP   0;
      A     L 0.0;
      A(;
      L     "DOOR_EXTRACTOR_DB".TRA_SLOW_FWD_OP_CT_TM;
      L     1;
      >=I;
      );
      =     "DOOR_EXTRACTOR_DB".TRA_SLOW_FWD_OP_CUT;
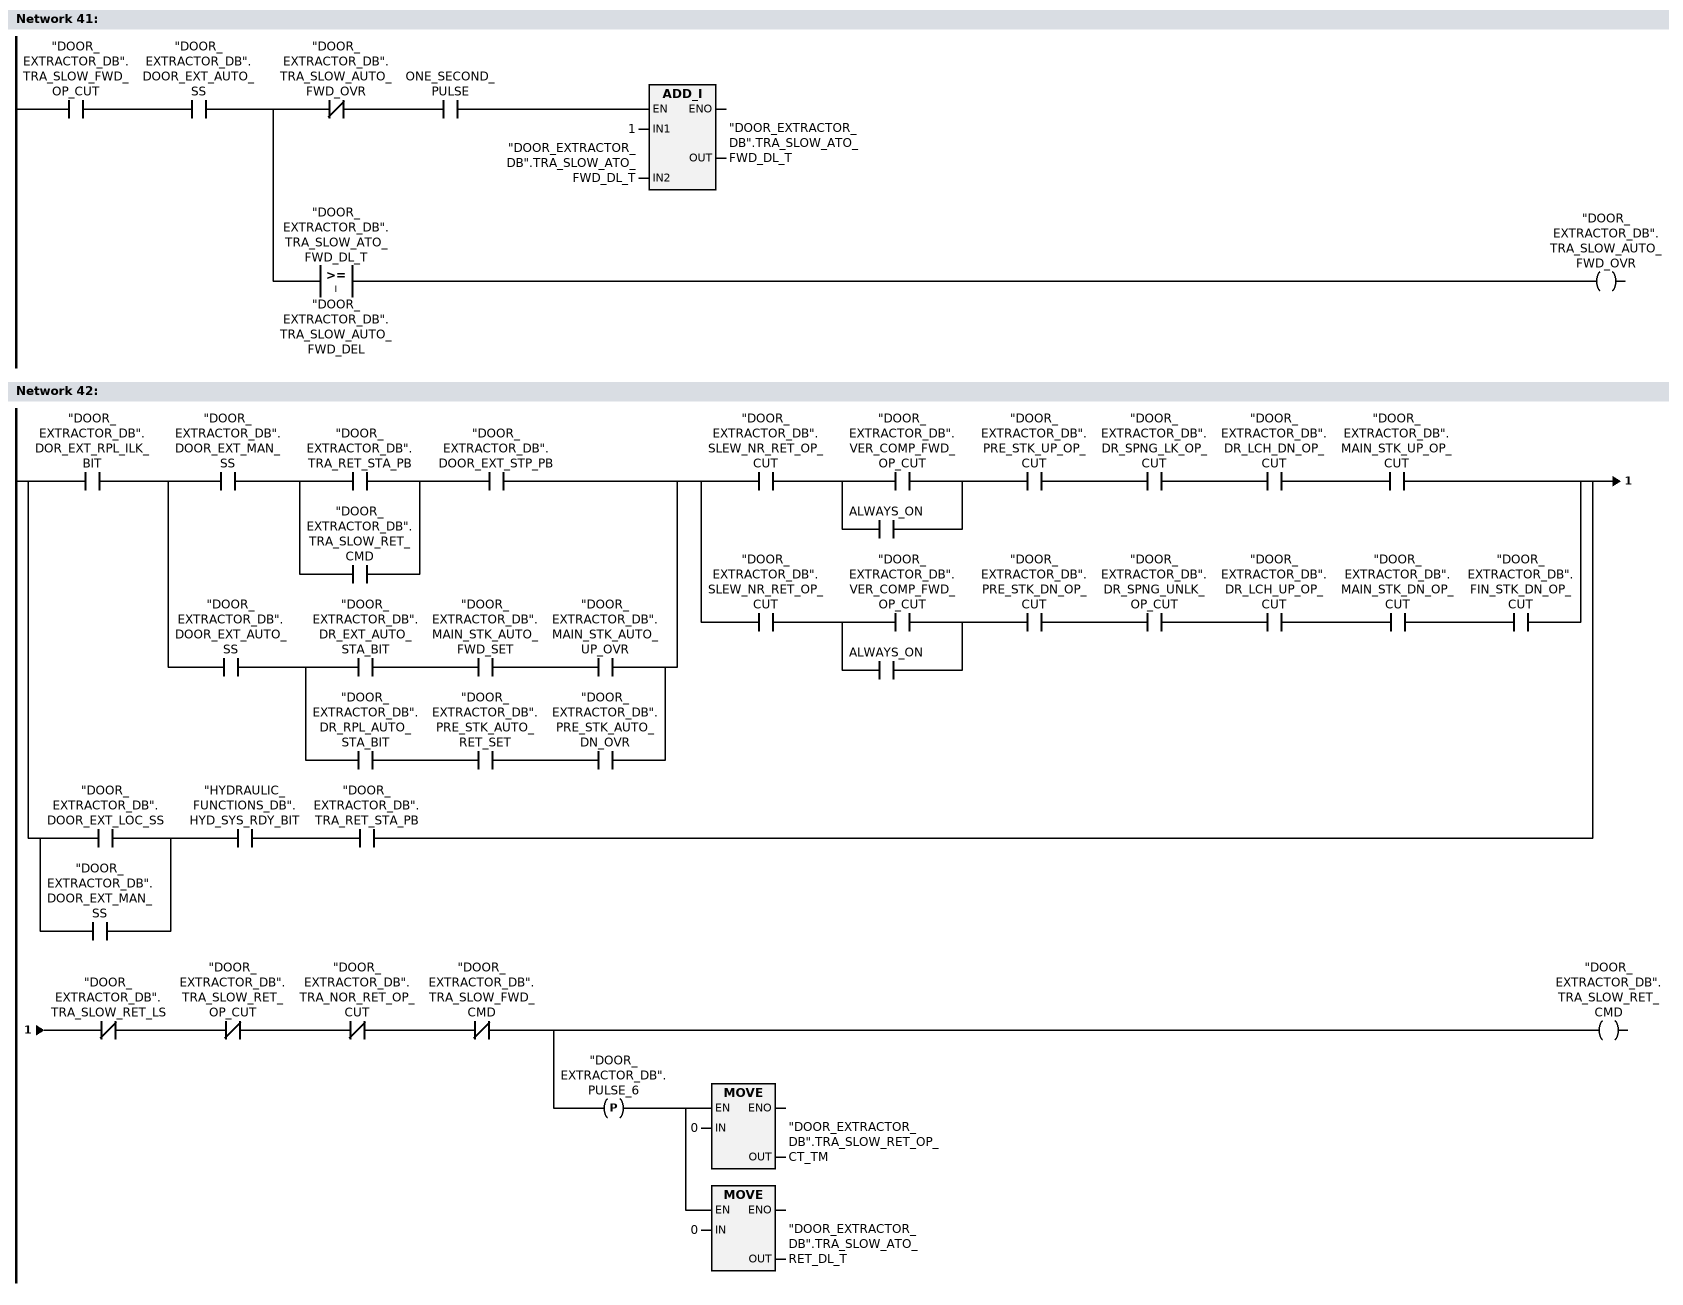
NETWORK
TITLE =
      A     "DOOR_EXTRACTOR_DB".TRA_SLOW_FWD_OP_CUT;
      A     "DOOR_EXTRACTOR_DB".DOOR_EXT_AUTO_SS;
      =     L 0.0;
      A     L 0.0;
      AN    "DOOR_EXTRACTOR_DB".TRA_SLOW_AUTO_FWD_OVR;
      A     "ONE_SECOND_PULSE";
      JNB   _022;
      L     1;
      L     "DOOR_EXTRACTOR_DB".TRA_SLOW_ATO_FWD_DL_T;
      +I;
      T     "DOOR_EXTRACTOR_DB".TRA_SLOW_ATO_FWD_DL_T;
_022: NOP   0;
      A     L 0.0;
      A(;
      L     "DOOR_EXTRACTOR_DB".TRA_SLOW_ATO_FWD_DL_T;
      L     "DOOR_EXTRACTOR_DB".TRA_SLOW_AUTO_FWD_DEL;
      >=I;
      );
      =     "DOOR_EXTRACTOR_DB".TRA_SLOW_AUTO_FWD_OVR;
NETWORK
TITLE =
      A(;
      A     "DOOR_EXTRACTOR_DB".DOR_EXT_RPL_ILK_BIT;
      A(;
      A     "DOOR_EXTRACTOR_DB".DOOR_EXT_MAN_SS;
      A(;
      O     "DOOR_EXTRACTOR_DB".TRA_RET_STA_PB;
      O     "DOOR_EXTRACTOR_DB".TRA_SLOW_RET_CMD;
      );
      A     "DOOR_EXTRACTOR_DB".DOOR_EXT_STP_PB;
      O;
      A     "DOOR_EXTRACTOR_DB".DOOR_EXT_AUTO_SS;
      A(;
      A     "DOOR_EXTRACTOR_DB".DR_EXT_AUTO_STA_BIT;
      A     "DOOR_EXTRACTOR_DB".MAIN_STK_AUTO_FWD_SET;
      A     "DOOR_EXTRACTOR_DB".MAIN_STK_AUTO_UP_OVR;
      O;
      A     "DOOR_EXTRACTOR_DB".DR_RPL_AUTO_STA_BIT;
      A     "DOOR_EXTRACTOR_DB".PRE_STK_AUTO_RET_SET;
      A     "DOOR_EXTRACTOR_DB".PRE_STK_AUTO_DN_OVR;
      );
      );
      A(;
      A     "DOOR_EXTRACTOR_DB".SLEW_NR_RET_OP_CUT;
      A(;
      O     "DOOR_EXTRACTOR_DB".VER_COMP_FWD_OP_CUT;
      O     "ALWAYS_ON";
      );
      A     "DOOR_EXTRACTOR_DB".PRE_STK_UP_OP_CUT;
      A     "DOOR_EXTRACTOR_DB".DR_SPNG_LK_OP_CUT;
      A     "DOOR_EXTRACTOR_DB".DR_LCH_DN_OP_CUT;
      A     "DOOR_EXTRACTOR_DB".MAIN_STK_UP_OP_CUT;
      O;
      A     "DOOR_EXTRACTOR_DB".SLEW_NR_RET_OP_CUT;
      A(;
      O     "DOOR_EXTRACTOR_DB".VER_COMP_FWD_OP_CUT;
      O     "ALWAYS_ON";
      );
      A     "DOOR_EXTRACTOR_DB".PRE_STK_DN_OP_CUT;
      A     "DOOR_EXTRACTOR_DB".DR_SPNG_UNLK_OP_CUT;
      A     "DOOR_EXTRACTOR_DB".DR_LCH_UP_OP_CUT;
      A     "DOOR_EXTRACTOR_DB".MAIN_STK_DN_OP_CUT;
      A     "DOOR_EXTRACTOR_DB".FIN_STK_DN_OP_CUT;
      );
      O;
      A(;
      O     "DOOR_EXTRACTOR_DB".DOOR_EXT_LOC_SS;
      O     "DOOR_EXTRACTOR_DB".DOOR_EXT_MAN_SS;
      );
      A     "HYDRAULIC_FUNCTIONS_DB".HYD_SYS_RDY_BIT;
      A     "DOOR_EXTRACTOR_DB".TRA_RET_STA_PB;
      );
      AN    "DOOR_EXTRACTOR_DB".TRA_SLOW_RET_LS;
      AN    "DOOR_EXTRACTOR_DB".TRA_SLOW_RET_OP_CUT;
      AN    "DOOR_EXTRACTOR_DB".TRA_NOR_RET_OP_CUT;
      AN    "DOOR_EXTRACTOR_DB".TRA_SLOW_FWD_CMD;
      =     L 0.0;
      A     L 0.0;
      BLD   102;
      =     "DOOR_EXTRACTOR_DB".TRA_SLOW_RET_CMD;
      A     L 0.0;
      FP    "DOOR_EXTRACTOR_DB".PULSE_6;
      =     L 0.1;
      A     L 0.1;
      JNB   _023;
      L     0;
      T     "DOOR_EXTRACTOR_DB".TRA_SLOW_RET_OP_CT_TM;
_023: NOP   0;
      A     L 0.1;
      JNB   _024;
      L     0;
      T     "DOOR_EXTRACTOR_DB".TRA_SLOW_ATO_RET_DL_T;
_024: NOP   0;
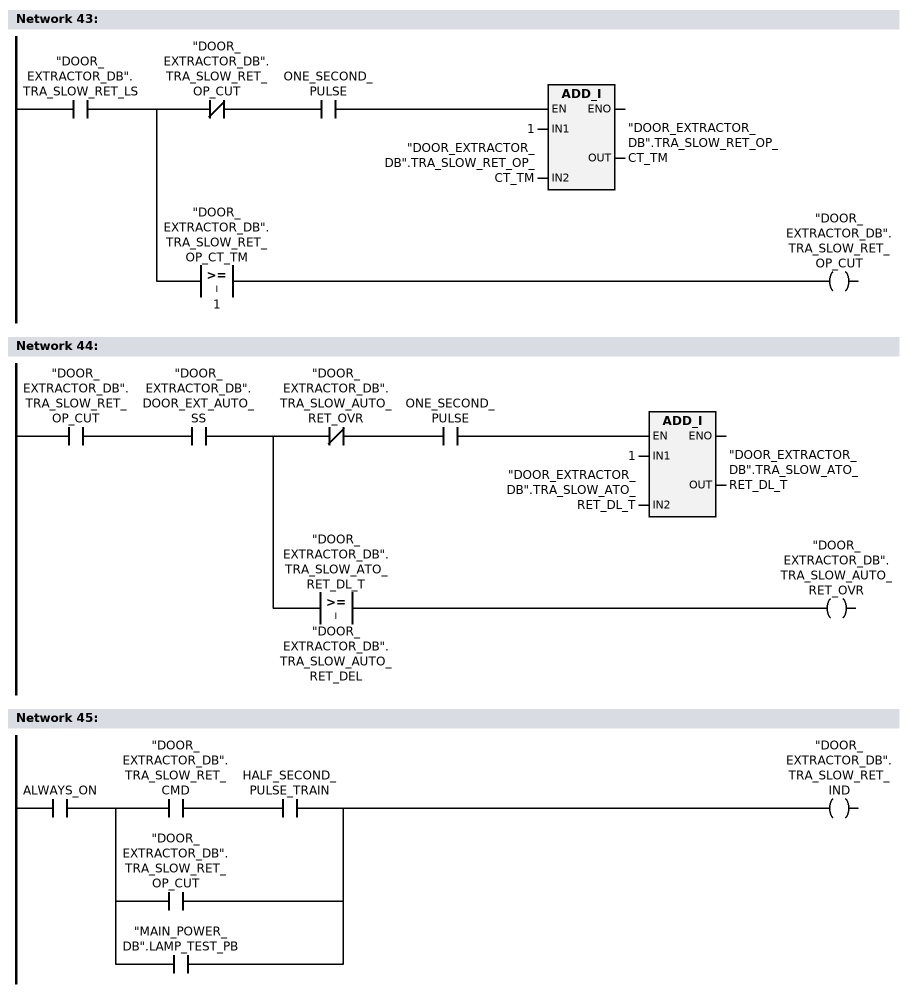
NETWORK
TITLE =
      A     "DOOR_EXTRACTOR_DB".TRA_SLOW_RET_LS;
      =     L 0.0;
      A     L 0.0;
      AN    "DOOR_EXTRACTOR_DB".TRA_SLOW_RET_OP_CUT;
      A     "ONE_SECOND_PULSE";
      JNB   _025;
      L     1;
      L     "DOOR_EXTRACTOR_DB".TRA_SLOW_RET_OP_CT_TM;
      +I;
      T     "DOOR_EXTRACTOR_DB".TRA_SLOW_RET_OP_CT_TM;
_025: NOP   0;
      A     L 0.0;
      A(;
      L     "DOOR_EXTRACTOR_DB".TRA_SLOW_RET_OP_CT_TM;
      L     1;
      >=I;
      );
      =     "DOOR_EXTRACTOR_DB".TRA_SLOW_RET_OP_CUT;
NETWORK
TITLE =
      A     "DOOR_EXTRACTOR_DB".TRA_SLOW_RET_OP_CUT;
      A     "DOOR_EXTRACTOR_DB".DOOR_EXT_AUTO_SS;
      =     L 0.0;
      A     L 0.0;
      AN    "DOOR_EXTRACTOR_DB".TRA_SLOW_AUTO_RET_OVR;
      A     "ONE_SECOND_PULSE";
      JNB   _026;
      L     1;
      L     "DOOR_EXTRACTOR_DB".TRA_SLOW_ATO_RET_DL_T;
      +I;
      T     "DOOR_EXTRACTOR_DB".TRA_SLOW_ATO_RET_DL_T;
_026: NOP   0;
      A     L 0.0;
      A(;
      L     "DOOR_EXTRACTOR_DB".TRA_SLOW_ATO_RET_DL_T;
      L     "DOOR_EXTRACTOR_DB".TRA_SLOW_AUTO_RET_DEL;
      >=I;
      );
      =     "DOOR_EXTRACTOR_DB".TRA_SLOW_AUTO_RET_OVR;
NETWORK
TITLE =
      A     "ALWAYS_ON";
      A(;
      A     "DOOR_EXTRACTOR_DB".TRA_SLOW_RET_CMD;
      A     "HALF_SECOND_PULSE_TRAIN";
      O     "DOOR_EXTRACTOR_DB".TRA_SLOW_RET_OP_CUT;
      O     "MAIN_POWER_DB".LAMP_TEST_PB;
      );
      =     "DOOR_EXTRACTOR_DB".TRA_SLOW_RET_IND;
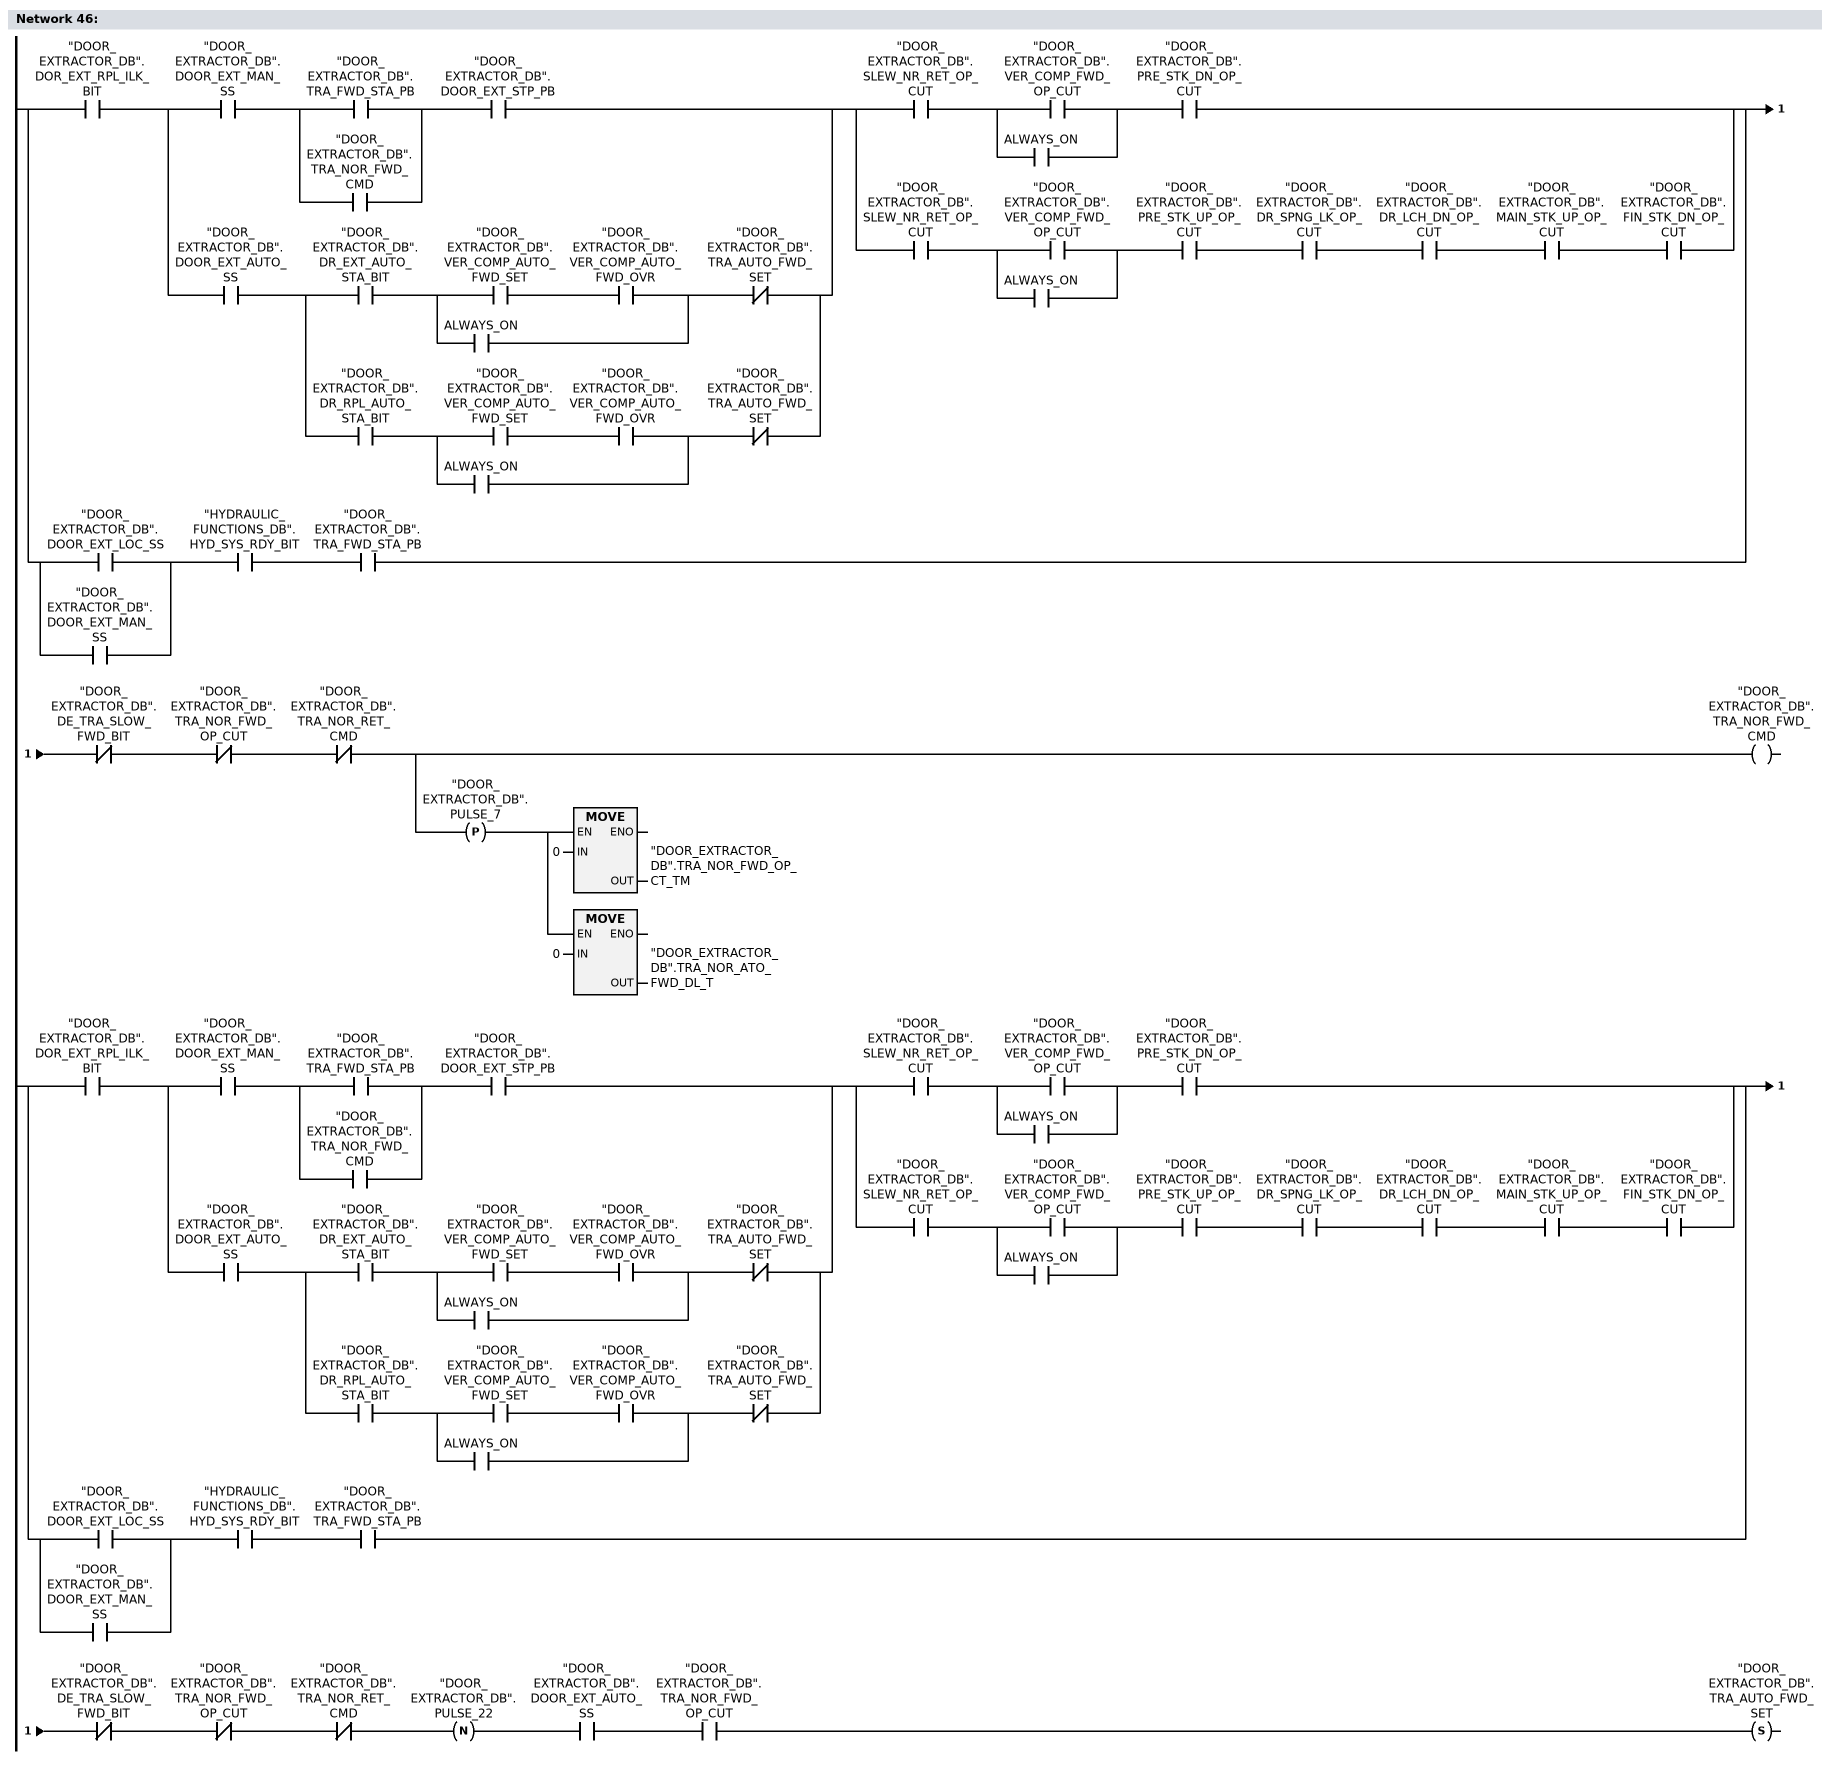
NETWORK
TITLE =
      A(;
      A     "DOOR_EXTRACTOR_DB".DOR_EXT_RPL_ILK_BIT;
      A(;
      A     "DOOR_EXTRACTOR_DB".DOOR_EXT_MAN_SS;
      A(;
      O     "DOOR_EXTRACTOR_DB".TRA_FWD_STA_PB;
      O     "DOOR_EXTRACTOR_DB".TRA_NOR_FWD_CMD;
      );
      A     "DOOR_EXTRACTOR_DB".DOOR_EXT_STP_PB;
      O;
      A     "DOOR_EXTRACTOR_DB".DOOR_EXT_AUTO_SS;
      A(;
      A     "DOOR_EXTRACTOR_DB".DR_EXT_AUTO_STA_BIT;
      A(;
      A     "DOOR_EXTRACTOR_DB".VER_COMP_AUTO_FWD_SET;
      A     "DOOR_EXTRACTOR_DB".VER_COMP_AUTO_FWD_OVR;
      O     "ALWAYS_ON";
      );
      AN    "DOOR_EXTRACTOR_DB".TRA_AUTO_FWD_SET;
      O;
      A     "DOOR_EXTRACTOR_DB".DR_RPL_AUTO_STA_BIT;
      A(;
      A     "DOOR_EXTRACTOR_DB".VER_COMP_AUTO_FWD_SET;
      A     "DOOR_EXTRACTOR_DB".VER_COMP_AUTO_FWD_OVR;
      O     "ALWAYS_ON";
      );
      AN    "DOOR_EXTRACTOR_DB".TRA_AUTO_FWD_SET;
      );
      );
      A(;
      A     "DOOR_EXTRACTOR_DB".SLEW_NR_RET_OP_CUT;
      A(;
      O     "DOOR_EXTRACTOR_DB".VER_COMP_FWD_OP_CUT;
      O     "ALWAYS_ON";
      );
      A     "DOOR_EXTRACTOR_DB".PRE_STK_DN_OP_CUT;
      O;
      A     "DOOR_EXTRACTOR_DB".SLEW_NR_RET_OP_CUT;
      A(;
      O     "DOOR_EXTRACTOR_DB".VER_COMP_FWD_OP_CUT;
      O     "ALWAYS_ON";
      );
      A     "DOOR_EXTRACTOR_DB".PRE_STK_UP_OP_CUT;
      A     "DOOR_EXTRACTOR_DB".DR_SPNG_LK_OP_CUT;
      A     "DOOR_EXTRACTOR_DB".DR_LCH_DN_OP_CUT;
      A     "DOOR_EXTRACTOR_DB".MAIN_STK_UP_OP_CUT;
      A     "DOOR_EXTRACTOR_DB".FIN_STK_DN_OP_CUT;
      );
      O;
      A(;
      O     "DOOR_EXTRACTOR_DB".DOOR_EXT_LOC_SS;
      O     "DOOR_EXTRACTOR_DB".DOOR_EXT_MAN_SS;
      );
      A     "HYDRAULIC_FUNCTIONS_DB".HYD_SYS_RDY_BIT;
      A     "DOOR_EXTRACTOR_DB".TRA_FWD_STA_PB;
      );
      AN    "DOOR_EXTRACTOR_DB".DE_TRA_SLOW_FWD_BIT;
      AN    "DOOR_EXTRACTOR_DB".TRA_NOR_FWD_OP_CUT;
      AN    "DOOR_EXTRACTOR_DB".TRA_NOR_RET_CMD;
      =     L 0.0;
      A     L 0.0;
      BLD   102;
      =     "DOOR_EXTRACTOR_DB".TRA_NOR_FWD_CMD;
      A(;
      A     L 0.0;
      FN    "DOOR_EXTRACTOR_DB".PULSE_22;
      );
      A     "DOOR_EXTRACTOR_DB".DOOR_EXT_AUTO_SS;
      A     "DOOR_EXTRACTOR_DB".TRA_NOR_FWD_OP_CUT;
      S     "DOOR_EXTRACTOR_DB".TRA_AUTO_FWD_SET;
      A     L 0.0;
      FP    "DOOR_EXTRACTOR_DB".PULSE_7;
      =     L 0.1;
      A     L 0.1;
      JNB   _027;
      L     0;
      T     "DOOR_EXTRACTOR_DB".TRA_NOR_FWD_OP_CT_TM;
_027: NOP   0;
      A     L 0.1;
      JNB   _028;
      L     0;
      T     "DOOR_EXTRACTOR_DB".TRA_NOR_ATO_FWD_DL_T;
_028: NOP   0;
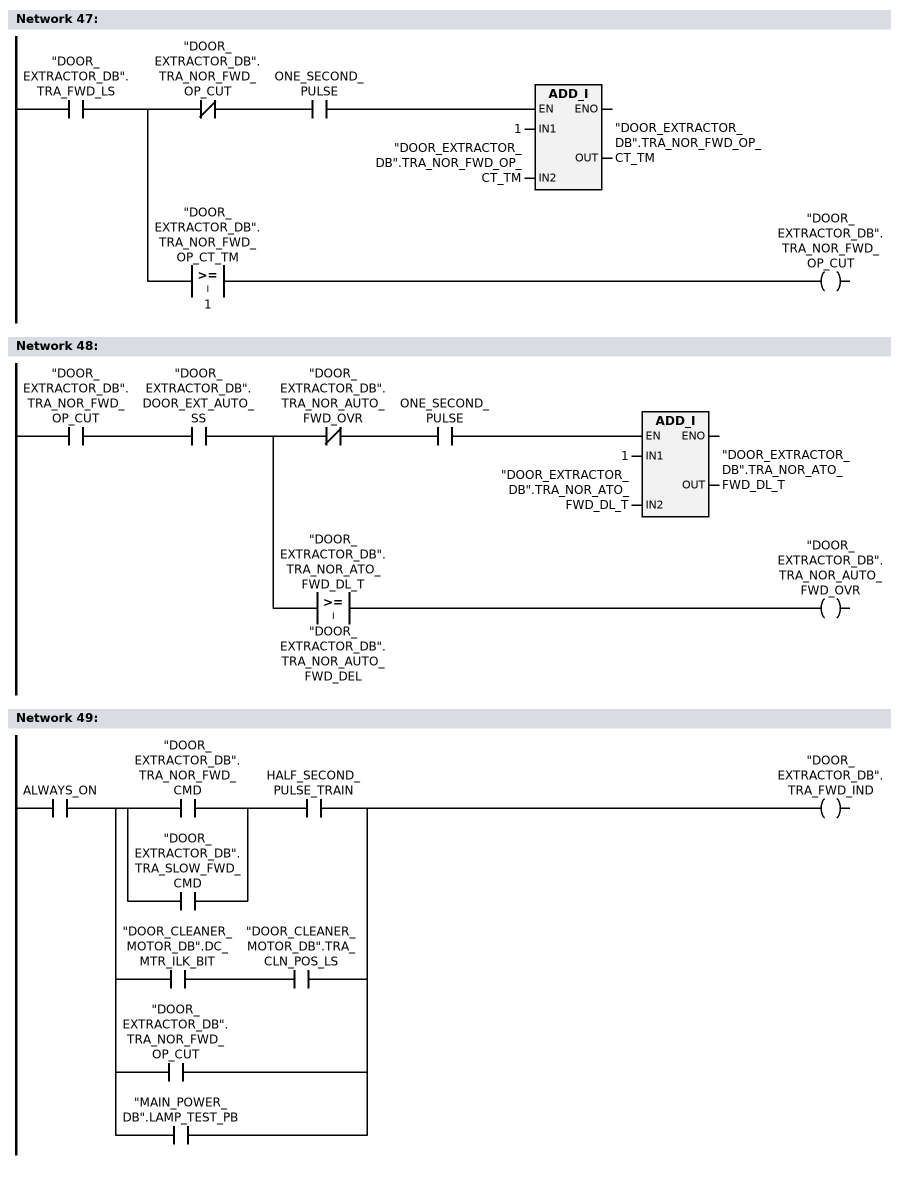
NETWORK
TITLE =
      A     "DOOR_EXTRACTOR_DB".TRA_FWD_LS;
      =     L 0.0;
      A     L 0.0;
      AN    "DOOR_EXTRACTOR_DB".TRA_NOR_FWD_OP_CUT;
      A     "ONE_SECOND_PULSE";
      JNB   _029;
      L     1;
      L     "DOOR_EXTRACTOR_DB".TRA_NOR_FWD_OP_CT_TM;
      +I;
      T     "DOOR_EXTRACTOR_DB".TRA_NOR_FWD_OP_CT_TM;
_029: NOP   0;
      A     L 0.0;
      A(;
      L     "DOOR_EXTRACTOR_DB".TRA_NOR_FWD_OP_CT_TM;
      L     1;
      >=I;
      );
      =     "DOOR_EXTRACTOR_DB".TRA_NOR_FWD_OP_CUT;
NETWORK
TITLE =
      A     "DOOR_EXTRACTOR_DB".TRA_NOR_FWD_OP_CUT;
      A     "DOOR_EXTRACTOR_DB".DOOR_EXT_AUTO_SS;
      =     L 0.0;
      A     L 0.0;
      AN    "DOOR_EXTRACTOR_DB".TRA_NOR_AUTO_FWD_OVR;
      A     "ONE_SECOND_PULSE";
      JNB   _02a;
      L     1;
      L     "DOOR_EXTRACTOR_DB".TRA_NOR_ATO_FWD_DL_T;
      +I;
      T     "DOOR_EXTRACTOR_DB".TRA_NOR_ATO_FWD_DL_T;
_02a: NOP   0;
      A     L 0.0;
      A(;
      L     "DOOR_EXTRACTOR_DB".TRA_NOR_ATO_FWD_DL_T;
      L     "DOOR_EXTRACTOR_DB".TRA_NOR_AUTO_FWD_DEL;
      >=I;
      );
      =     "DOOR_EXTRACTOR_DB".TRA_NOR_AUTO_FWD_OVR;
NETWORK
TITLE =
      A     "ALWAYS_ON";
      A(;
      A(;
      O     "DOOR_EXTRACTOR_DB".TRA_NOR_FWD_CMD;
      O     "DOOR_EXTRACTOR_DB".TRA_SLOW_FWD_CMD;
      );
      A     "HALF_SECOND_PULSE_TRAIN";
      O;
      A     "DOOR_CLEANER_MOTOR_DB".DC_MTR_ILK_BIT;
      A     "DOOR_CLEANER_MOTOR_DB".TRA_CLN_POS_LS;
      O     "DOOR_EXTRACTOR_DB".TRA_NOR_FWD_OP_CUT;
      O     "MAIN_POWER_DB".LAMP_TEST_PB;
      );
      =     "DOOR_EXTRACTOR_DB".TRA_FWD_IND;
